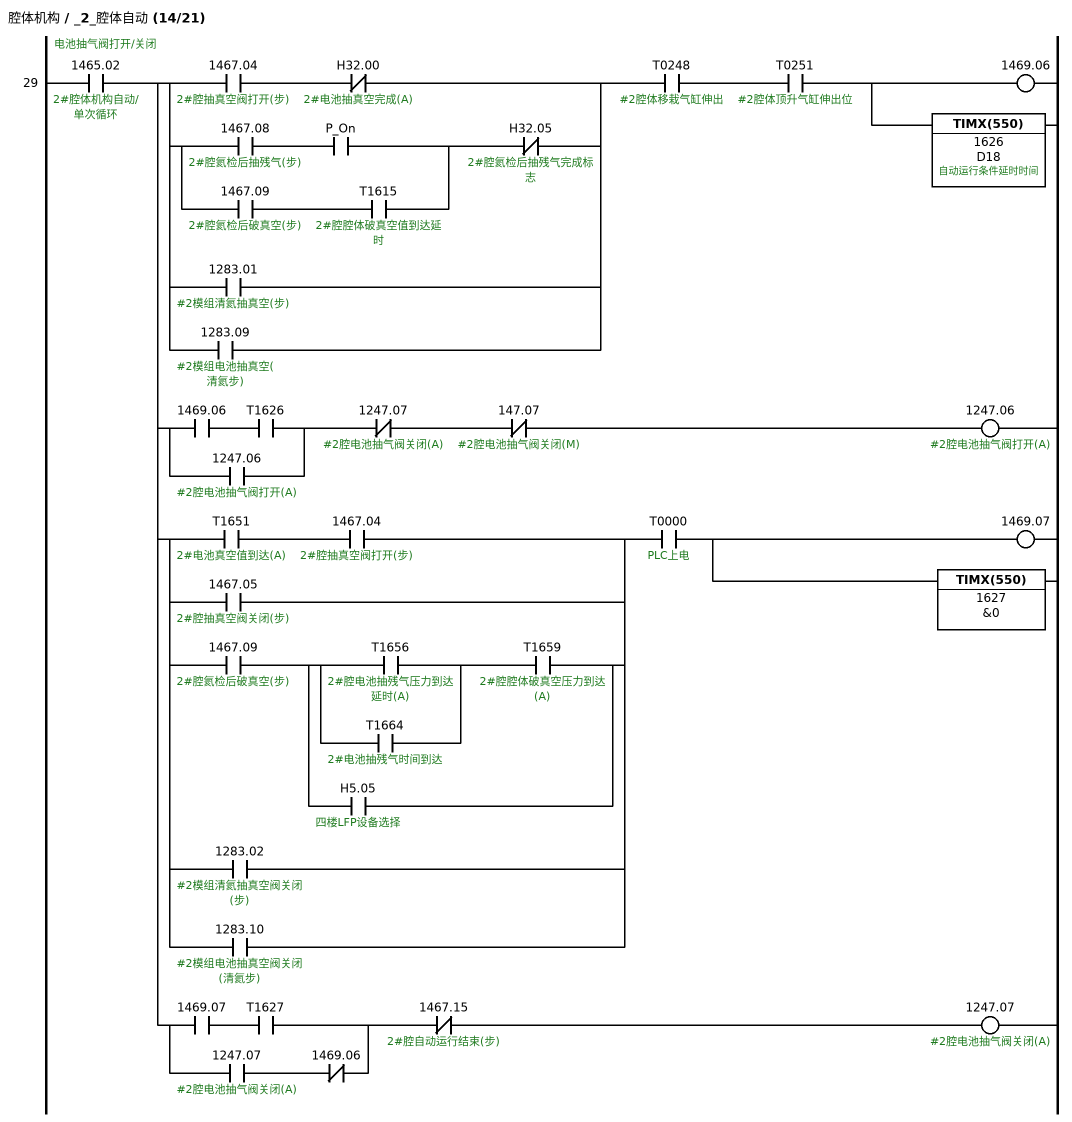
; [picture p312: 腔体机构 / _2_腔体自动, rungs 29-29]
; rung 29: 电池抽气阀打开/关闭
LD 1465.02  ; 2#腔体机构自动/单次循环
OUT TR0
LD 1467.04  ; 2#腔抽真空阀打开(步)
ANDNOT H32.00  ; 2#电池抽真空完成(A)
LD 1467.08  ; 2#腔氦检后抽残气(步)
AND P_On
LD 1467.09  ; 2#腔氦检后破真空(步)
AND T1615  ; 2#腔腔体破真空值到达延时
ORLD
ANDNOT H32.05  ; 2#腔氦检后抽残气完成标志
ORLD
OR 1283.01  ; #2模组清氦抽真空(步)
OR 1283.09  ; #2模组电池抽真空(清氦步)
ANDLD
AND T0248  ; #2腔体移栽气缸伸出
AND T0251  ; #2腔体顶升气缸伸出位
OUT 1469.06
TIMX(550) 1626 D18  ; 自动运行条件延时时间
LD TR0
LD 1469.06
AND T1626
OR 1247.06  ; #2腔电池抽气阀打开(A)
ANDLD
ANDNOT 1247.07  ; #2腔电池抽气阀关闭(A)
ANDNOT 147.07  ; #2腔电池抽气阀关闭(M)
OUT 1247.06  ; #2腔电池抽气阀打开(A)
LD TR0
LD T1651  ; 2#电池真空值到达(A)
AND 1467.04  ; 2#腔抽真空阀打开(步)
OR 1467.05  ; 2#腔抽真空阀关闭(步)
LD 1467.09  ; 2#腔氦检后破真空(步)
LD T1656  ; 2#腔电池抽残气压力到达延时(A)
OR T1664  ; 2#电池抽残气时间到达
AND T1659  ; 2#腔腔体破真空压力到达(A)
OR H5.05  ; 四楼LFP设备选择
ANDLD
ORLD
OR 1283.02  ; #2模组清氦抽真空阀关闭(步)
OR 1283.10  ; #2模组电池抽真空阀关闭(清氦步)
ANDLD
AND T0000  ; PLC上电
OUT 1469.07
TIMX(550) 1627 &0
LD TR0
LD 1469.07
AND T1627
LD 1247.07  ; #2腔电池抽气阀关闭(A)
ANDNOT 1469.06
ORLD
ANDLD
ANDNOT 1467.15  ; 2#腔自动运行结束(步)
OUT 1247.07  ; #2腔电池抽气阀关闭(A)

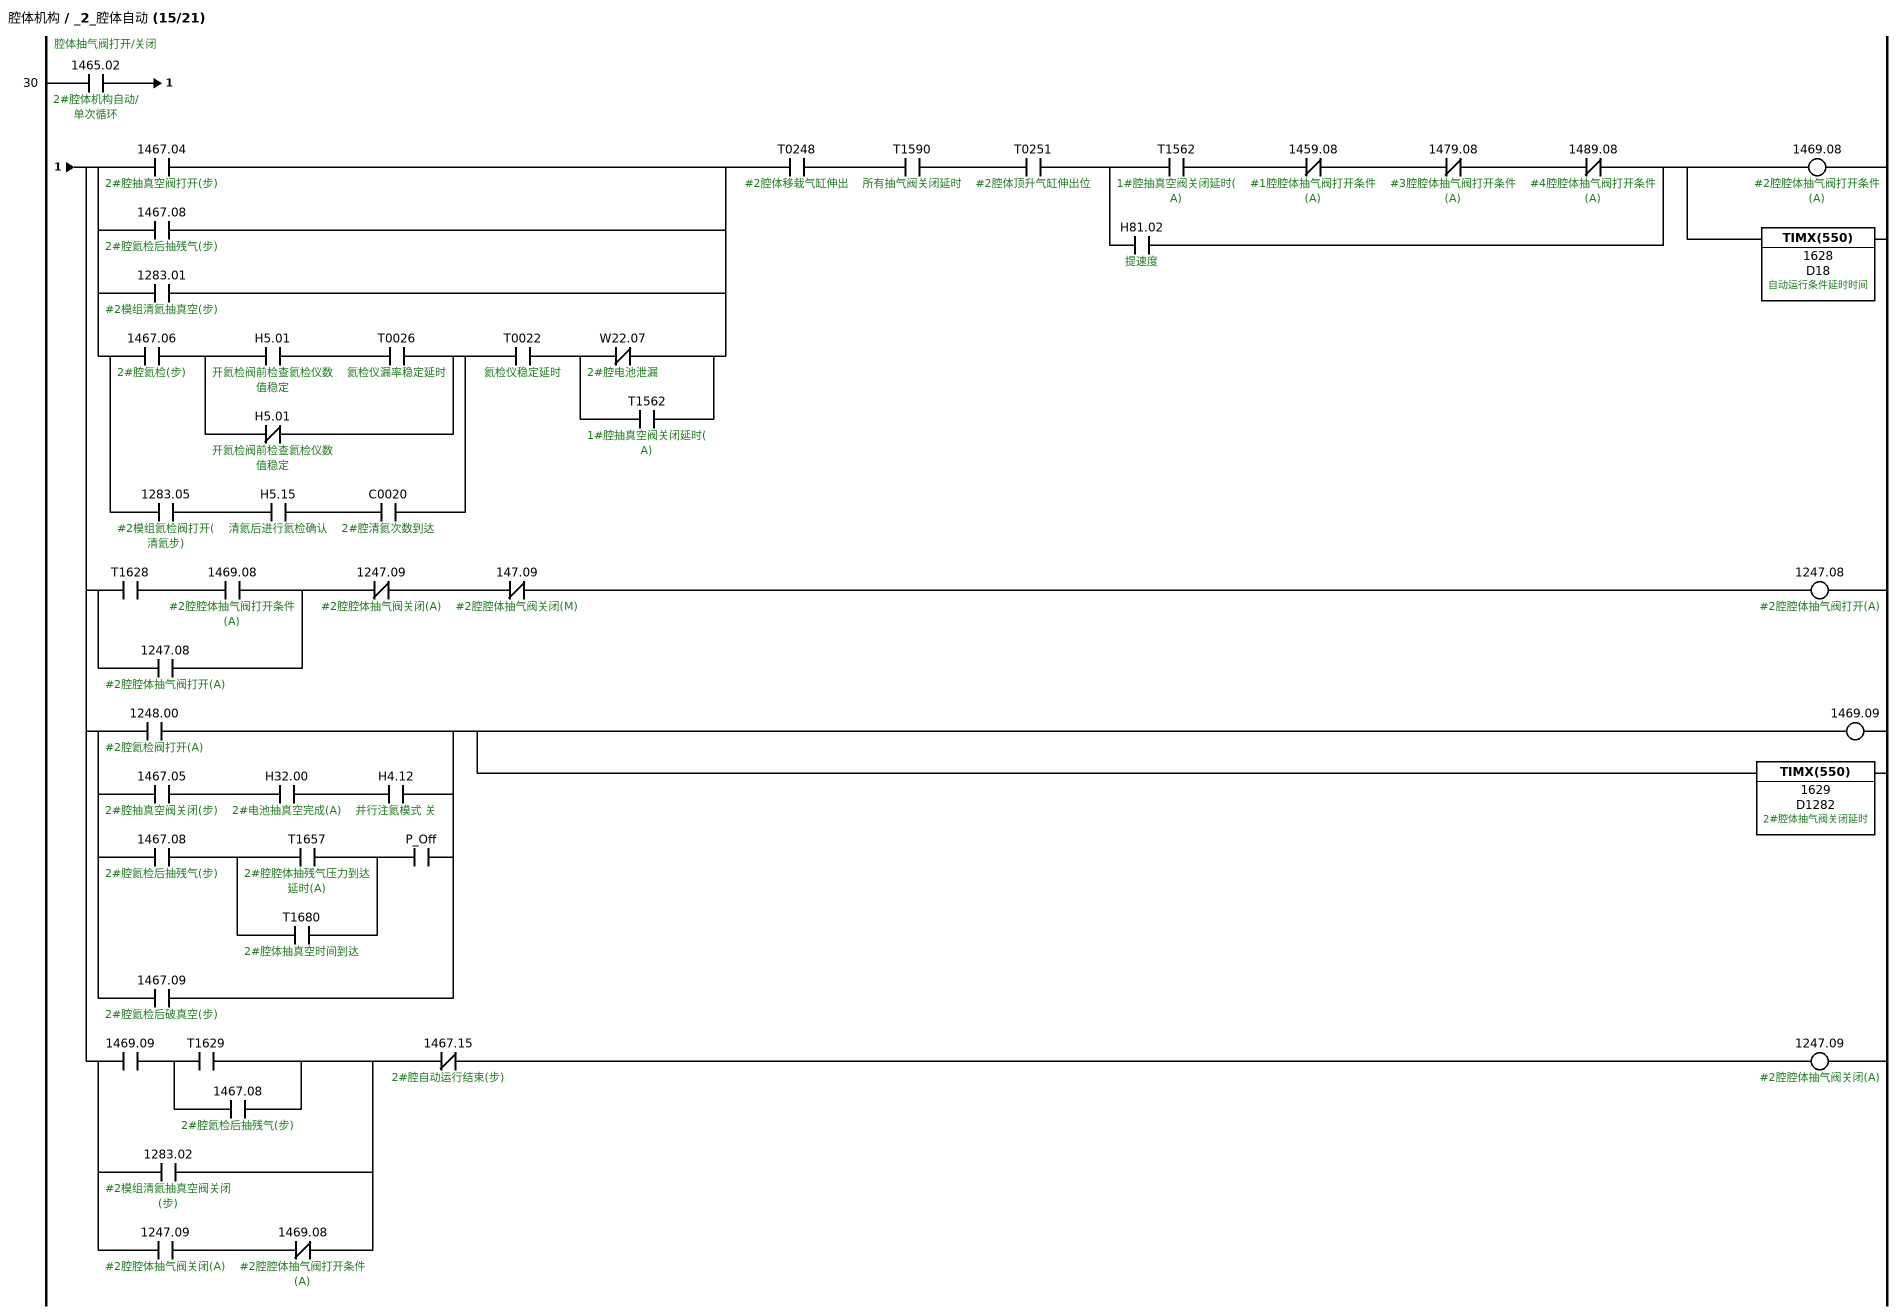
; rung 30: 腔体抽气阀打开/关闭
LD 1465.02  ; 2#腔体机构自动/单次循环
OUT TR0
LD 1467.04  ; 2#腔抽真空阀打开(步)
OR 1467.08  ; 2#腔氦检后抽残气(步)
OR 1283.01  ; #2模组清氦抽真空(步)
LD 1467.06  ; 2#腔氦检(步)
LD H5.01  ; 开氦检阀前检查氦检仪数值稳定
AND T0026  ; 氦检仪漏率稳定延时
ORNOT H5.01  ; 开氦检阀前检查氦检仪数值稳定
ANDLD
LD 1283.05  ; #2模组氦检阀打开(清氦步)
AND H5.15  ; 清氦后进行氦检确认
AND C0020  ; 2#腔清氦次数到达
ORLD
AND T0022  ; 氦检仪稳定延时
LDNOT W22.07  ; 2#腔电池泄漏
OR T1562  ; 1#腔抽真空阀关闭延时(A)
ANDLD
ORLD
ANDLD
AND T0248  ; #2腔体移栽气缸伸出
AND T1590  ; 所有抽气阀关闭延时
AND T0251  ; #2腔体顶升气缸伸出位
LD T1562  ; 1#腔抽真空阀关闭延时(A)
ANDNOT 1459.08  ; #1腔腔体抽气阀打开条件(A)
ANDNOT 1479.08  ; #3腔腔体抽气阀打开条件(A)
ANDNOT 1489.08  ; #4腔腔体抽气阀打开条件(A)
OR H81.02  ; 提速度
ANDLD
OUT 1469.08  ; #2腔腔体抽气阀打开条件(A)
TIMX(550) 1628 D18  ; 自动运行条件延时时间
LD TR0
LD T1628
AND 1469.08  ; #2腔腔体抽气阀打开条件(A)
OR 1247.08  ; #2腔腔体抽气阀打开(A)
ANDLD
ANDNOT 1247.09  ; #2腔腔体抽气阀关闭(A)
ANDNOT 147.09  ; #2腔腔体抽气阀关闭(M)
OUT 1247.08  ; #2腔腔体抽气阀打开(A)
LD TR0
LD 1248.00  ; #2腔氦检阀打开(A)
LD 1467.05  ; 2#腔抽真空阀关闭(步)
AND H32.00  ; 2#电池抽真空完成(A)
AND H4.12  ; 并行注氦模式 关
ORLD
LD 1467.08  ; 2#腔氦检后抽残气(步)
LD T1657  ; 2#腔腔体抽残气压力到达延时(A)
OR T1680  ; 2#腔体抽真空时间到达
ANDLD
AND P_Off
ORLD
OR 1467.09  ; 2#腔氦检后破真空(步)
ANDLD
OUT 1469.09
TIMX(550) 1629 D1282  ; 2#腔体抽气阀关闭延时
LD TR0
LD 1469.09
LD T1629
OR 1467.08  ; 2#腔氦检后抽残气(步)
ANDLD
OR 1283.02  ; #2模组清氦抽真空阀关闭(步)
LD 1247.09  ; #2腔腔体抽气阀关闭(A)
ANDNOT 1469.08  ; #2腔腔体抽气阀打开条件(A)
ORLD
ANDLD
ANDNOT 1467.15  ; 2#腔自动运行结束(步)
OUT 1247.09  ; #2腔腔体抽气阀关闭(A)

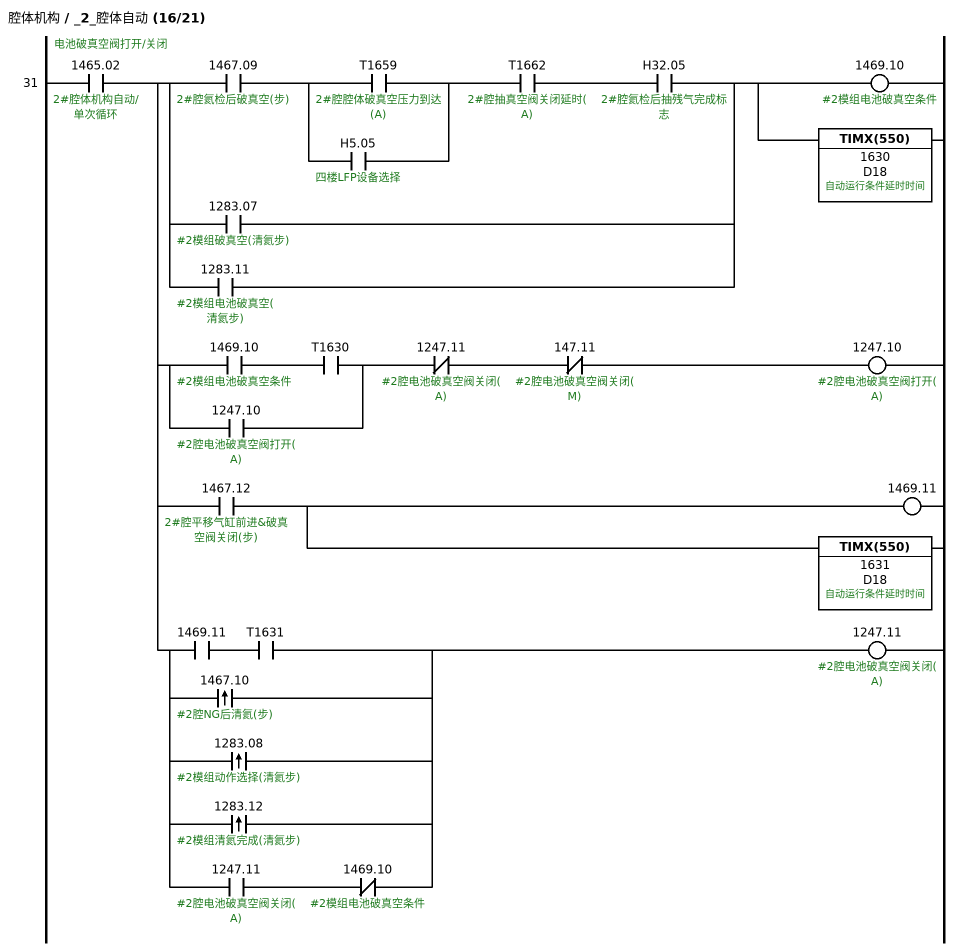
; rung 31: 电池破真空阀打开/关闭
LD 1465.02  ; 2#腔体机构自动/单次循环
OUT TR0
LD 1467.09  ; 2#腔氦检后破真空(步)
LD T1659  ; 2#腔腔体破真空压力到达(A)
OR H5.05  ; 四楼LFP设备选择
ANDLD
AND T1662  ; 2#腔抽真空阀关闭延时(A)
AND H32.05  ; 2#腔氦检后抽残气完成标志
OR 1283.07  ; #2模组破真空(清氦步)
OR 1283.11  ; #2模组电池破真空(清氦步)
ANDLD
OUT 1469.10  ; #2模组电池破真空条件
TIMX(550) 1630 D18  ; 自动运行条件延时时间
LD TR0
LD 1469.10  ; #2模组电池破真空条件
AND T1630
OR 1247.10  ; #2腔电池破真空阀打开(A)
ANDLD
ANDNOT 1247.11  ; #2腔电池破真空阀关闭(A)
ANDNOT 147.11  ; #2腔电池破真空阀关闭(M)
OUT 1247.10  ; #2腔电池破真空阀打开(A)
LD TR0
AND 1467.12  ; 2#腔平移气缸前进&破真空阀关闭(步)
OUT 1469.11
TIMX(550) 1631 D18  ; 自动运行条件延时时间
LD TR0
LD 1469.11
AND T1631
@OR 1467.10  ; #2腔NG后清氦(步)
@OR 1283.08  ; #2模组动作选择(清氦步)
@OR 1283.12  ; #2模组清氦完成(清氦步)
LD 1247.11  ; #2腔电池破真空阀关闭(A)
ANDNOT 1469.10  ; #2模组电池破真空条件
ORLD
ANDLD
OUT 1247.11  ; #2腔电池破真空阀关闭(A)

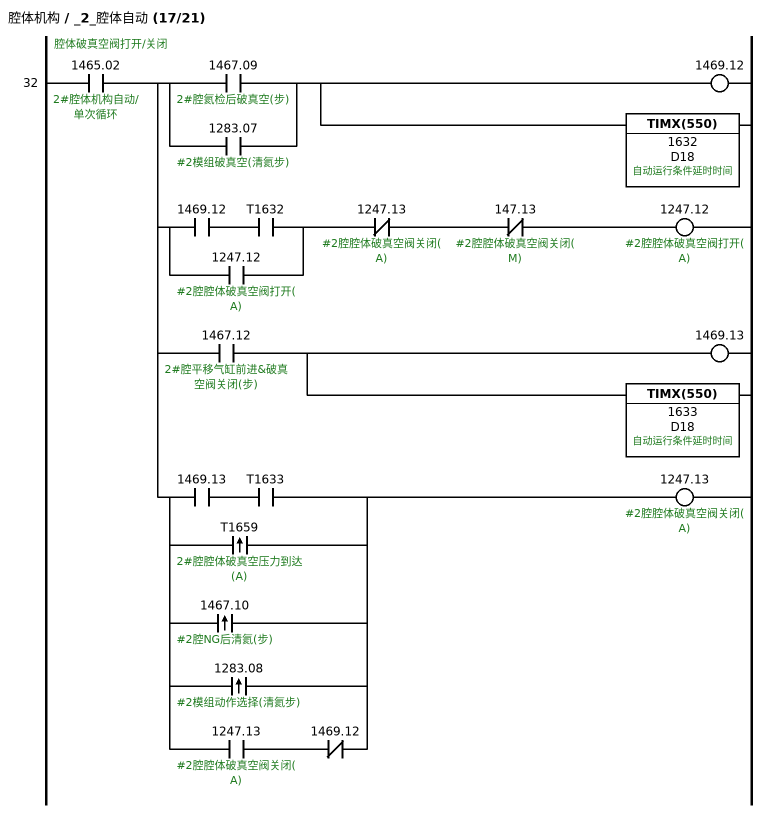
; rung 32: 腔体破真空阀打开/关闭
LD 1465.02  ; 2#腔体机构自动/单次循环
OUT TR0
LD 1467.09  ; 2#腔氦检后破真空(步)
OR 1283.07  ; #2模组破真空(清氦步)
ANDLD
OUT 1469.12
TIMX(550) 1632 D18  ; 自动运行条件延时时间
LD TR0
LD 1469.12
AND T1632
OR 1247.12  ; #2腔腔体破真空阀打开(A)
ANDLD
ANDNOT 1247.13  ; #2腔腔体破真空阀关闭(A)
ANDNOT 147.13  ; #2腔腔体破真空阀关闭(M)
OUT 1247.12  ; #2腔腔体破真空阀打开(A)
LD TR0
AND 1467.12  ; 2#腔平移气缸前进&破真空阀关闭(步)
OUT 1469.13
TIMX(550) 1633 D18  ; 自动运行条件延时时间
LD TR0
LD 1469.13
AND T1633
@OR T1659  ; 2#腔腔体破真空压力到达(A)
@OR 1467.10  ; #2腔NG后清氦(步)
@OR 1283.08  ; #2模组动作选择(清氦步)
LD 1247.13  ; #2腔腔体破真空阀关闭(A)
ANDNOT 1469.12
ORLD
ANDLD
OUT 1247.13  ; #2腔腔体破真空阀关闭(A)

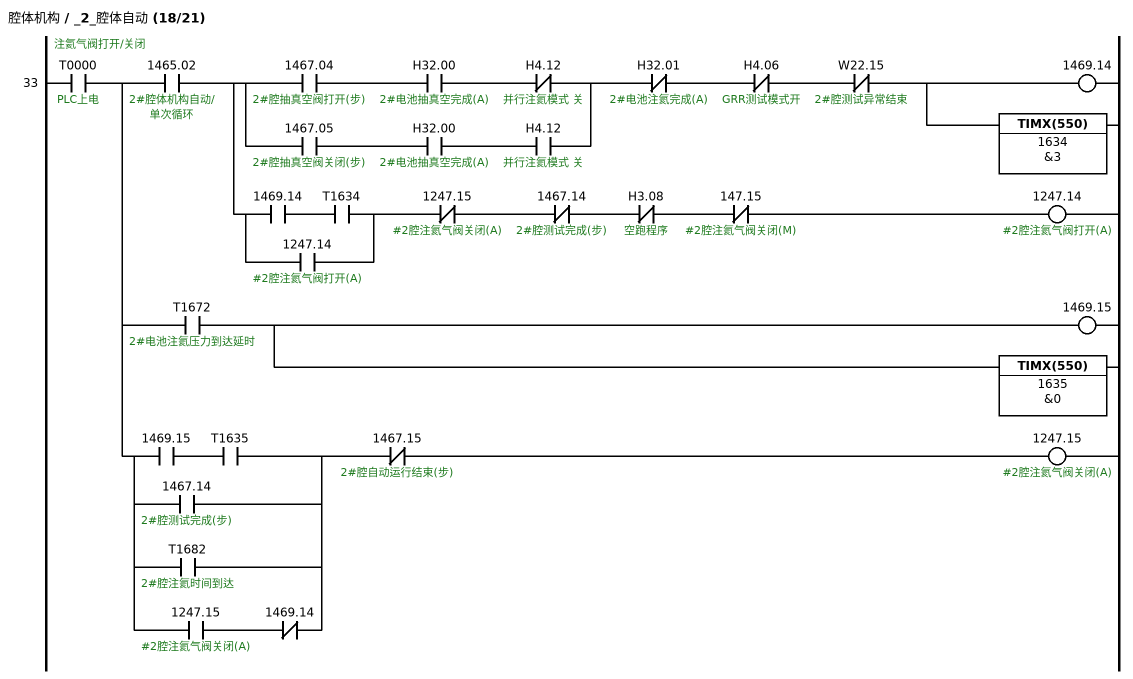
; rung 33: 注氦气阀打开/关闭
LD T0000  ; PLC上电
OUT TR0
AND 1465.02  ; 2#腔体机构自动/单次循环
OUT TR1
LD 1467.04  ; 2#腔抽真空阀打开(步)
AND H32.00  ; 2#电池抽真空完成(A)
ANDNOT H4.12  ; 并行注氦模式 关
LD 1467.05  ; 2#腔抽真空阀关闭(步)
AND H32.00  ; 2#电池抽真空完成(A)
AND H4.12  ; 并行注氦模式 关
ORLD
ANDLD
ANDNOT H32.01  ; 2#电池注氦完成(A)
ANDNOT H4.06  ; GRR测试模式开
ANDNOT W22.15  ; 2#腔测试异常结束
OUT 1469.14
TIMX(550) 1634 &3
LD TR1
LD 1469.14
AND T1634
OR 1247.14  ; #2腔注氦气阀打开(A)
ANDLD
ANDNOT 1247.15  ; #2腔注氦气阀关闭(A)
ANDNOT 1467.14  ; 2#腔测试完成(步)
ANDNOT H3.08  ; 空跑程序
ANDNOT 147.15  ; #2腔注氦气阀关闭(M)
OUT 1247.14  ; #2腔注氦气阀打开(A)
LD TR0
AND T1672  ; 2#电池注氦压力到达延时
OUT 1469.15
TIMX(550) 1635 &0
LD TR0
LD 1469.15
AND T1635
OR 1467.14  ; 2#腔测试完成(步)
OR T1682  ; 2#腔注氦时间到达
LD 1247.15  ; #2腔注氦气阀关闭(A)
ANDNOT 1469.14
ORLD
ANDLD
ANDNOT 1467.15  ; 2#腔自动运行结束(步)
OUT 1247.15  ; #2腔注氦气阀关闭(A)

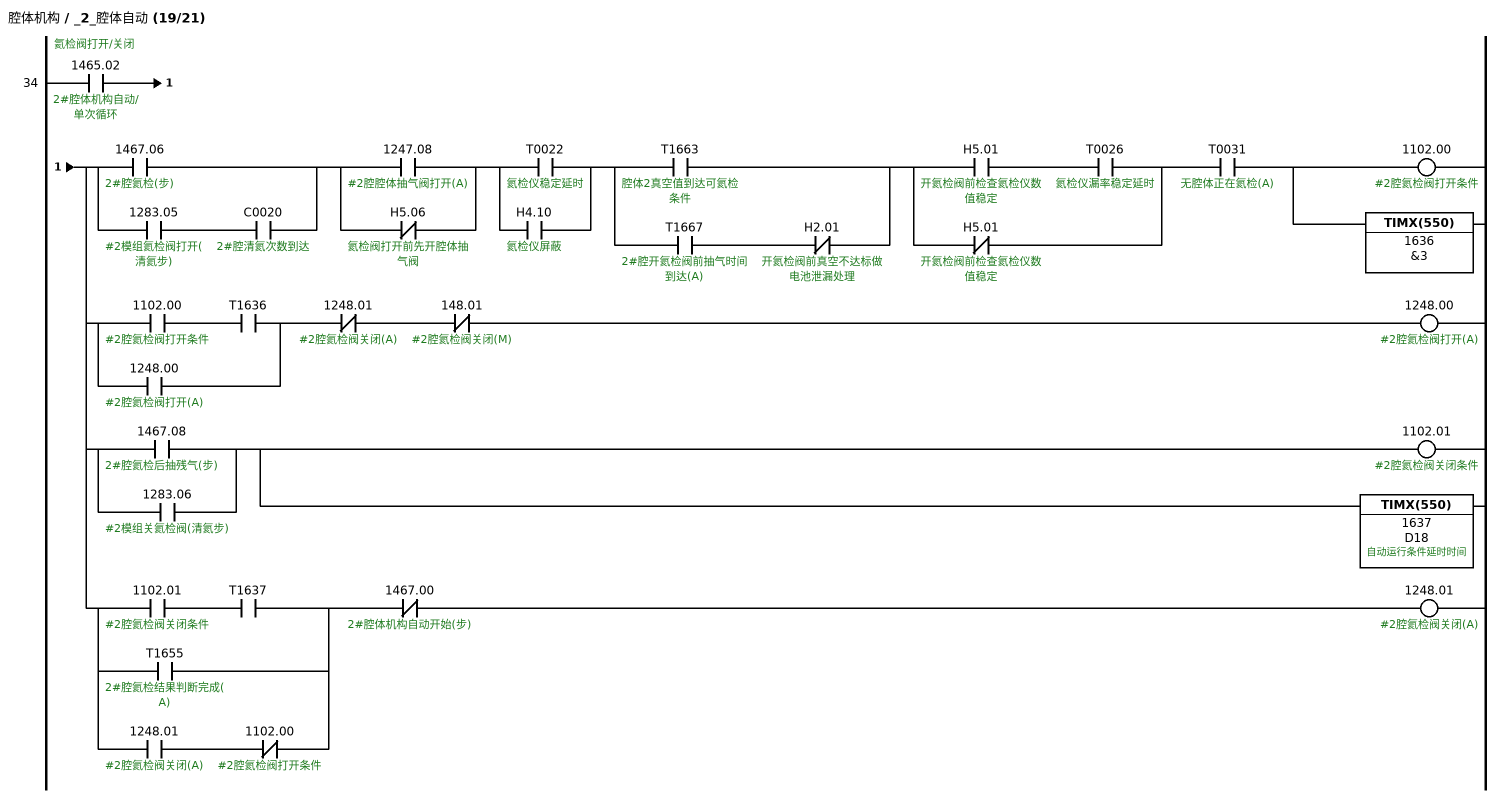
; rung 34: 氦检阀打开/关闭
LD 1465.02  ; 2#腔体机构自动/单次循环
OUT TR0
LD 1467.06  ; 2#腔氦检(步)
LD 1283.05  ; #2模组氦检阀打开(清氦步)
AND C0020  ; 2#腔清氦次数到达
ORLD
ANDLD
LD 1247.08  ; #2腔腔体抽气阀打开(A)
ORNOT H5.06  ; 氦检阀打开前先开腔体抽气阀
ANDLD
LD T0022  ; 氦检仪稳定延时
OR H4.10  ; 氦检仪屏蔽
ANDLD
LD T1663  ; 腔体2真空值到达可氦检条件
LD T1667  ; 2#腔开氦检阀前抽气时间到达(A)
ANDNOT H2.01  ; 开氦检阀前真空不达标做电池泄漏处理
ORLD
ANDLD
LD H5.01  ; 开氦检阀前检查氦检仪数值稳定
AND T0026  ; 氦检仪漏率稳定延时
ORNOT H5.01  ; 开氦检阀前检查氦检仪数值稳定
ANDLD
AND T0031  ; 无腔体正在氦检(A)
OUT 1102.00  ; #2腔氦检阀打开条件
TIMX(550) 1636 &3
LD TR0
LD 1102.00  ; #2腔氦检阀打开条件
AND T1636
OR 1248.00  ; #2腔氦检阀打开(A)
ANDLD
ANDNOT 1248.01  ; #2腔氦检阀关闭(A)
ANDNOT 148.01  ; #2腔氦检阀关闭(M)
OUT 1248.00  ; #2腔氦检阀打开(A)
LD TR0
LD 1467.08  ; 2#腔氦检后抽残气(步)
OR 1283.06  ; #2模组关氦检阀(清氦步)
ANDLD
OUT 1102.01  ; #2腔氦检阀关闭条件
TIMX(550) 1637 D18  ; 自动运行条件延时时间
LD TR0
LD 1102.01  ; #2腔氦检阀关闭条件
AND T1637
OR T1655  ; 2#腔氦检结果判断完成(A)
LD 1248.01  ; #2腔氦检阀关闭(A)
ANDNOT 1102.00  ; #2腔氦检阀打开条件
ORLD
ANDLD
ANDNOT 1467.00  ; 2#腔体机构自动开始(步)
OUT 1248.01  ; #2腔氦检阀关闭(A)

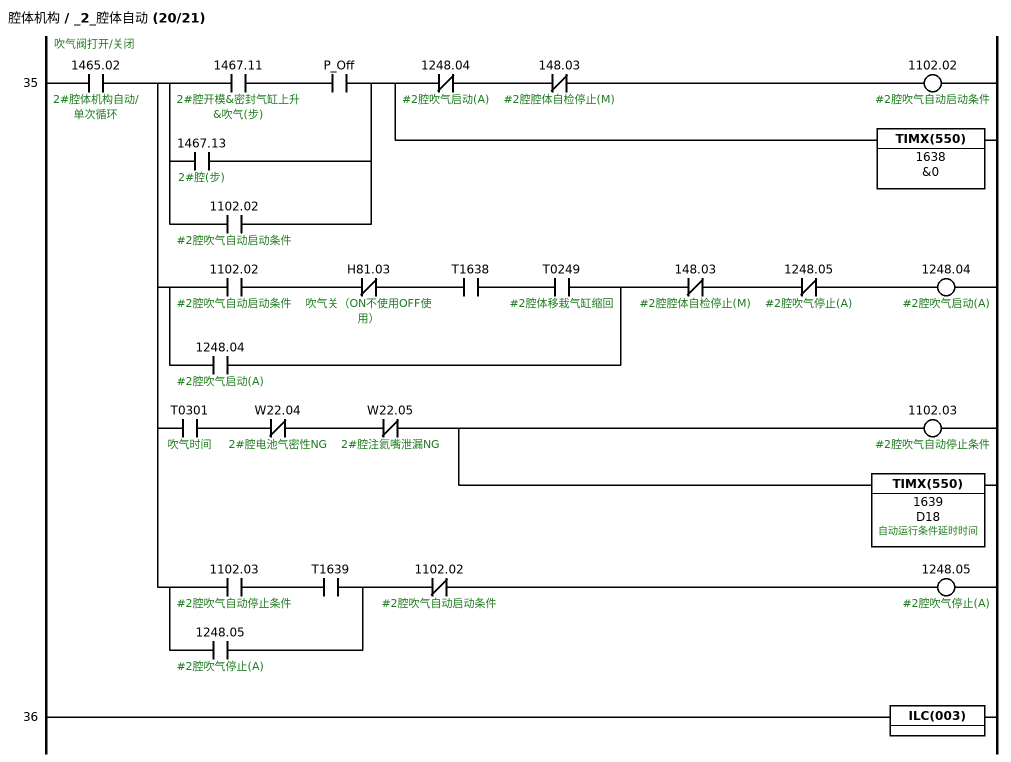
; rung 35: 吹气阀打开/关闭
LD 1465.02  ; 2#腔体机构自动/单次循环
OUT TR0
LD 1467.11  ; 2#腔开模&密封气缸上升&吹气(步)
AND P_Off
OR 1467.13  ; 2#腔(步)
OR 1102.02  ; #2腔吹气自动启动条件
ANDLD
OUT TR1
ANDNOT 1248.04  ; #2腔吹气启动(A)
ANDNOT 148.03  ; #2腔腔体自检停止(M)
OUT 1102.02  ; #2腔吹气自动启动条件
LD TR1
TIMX(550) 1638 &0
LD TR0
LD 1102.02  ; #2腔吹气自动启动条件
ANDNOT H81.03  ; 吹气关（ON不使用OFF使用）
AND T1638
AND T0249  ; #2腔体移栽气缸缩回
OR 1248.04  ; #2腔吹气启动(A)
ANDLD
ANDNOT 148.03  ; #2腔腔体自检停止(M)
ANDNOT 1248.05  ; #2腔吹气停止(A)
OUT 1248.04  ; #2腔吹气启动(A)
LD TR0
AND T0301  ; 吹气时间
ANDNOT W22.04  ; 2#腔电池气密性NG
ANDNOT W22.05  ; 2#腔注氦嘴泄漏NG
OUT 1102.03  ; #2腔吹气自动停止条件
TIMX(550) 1639 D18  ; 自动运行条件延时时间
LD TR0
LD 1102.03  ; #2腔吹气自动停止条件
AND T1639
OR 1248.05  ; #2腔吹气停止(A)
ANDLD
ANDNOT 1102.02  ; #2腔吹气自动启动条件
OUT 1248.05  ; #2腔吹气停止(A)
; rung 36
ILC(003)

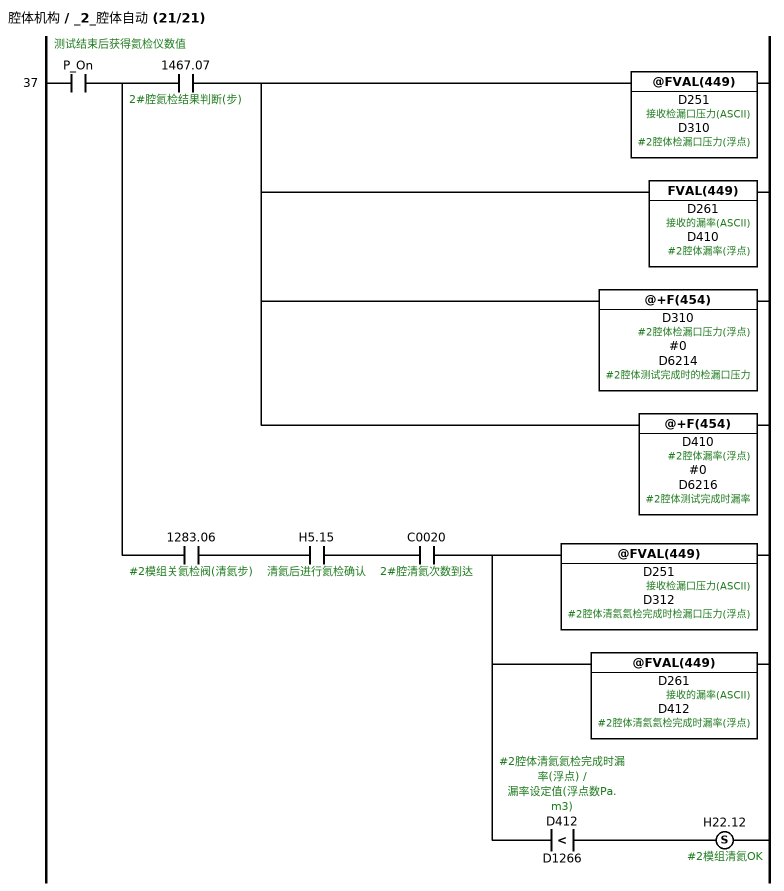
; rung 37: 测试结束后获得氦检仪数值
LD P_On
OUT TR0
AND 1467.07  ; 2#腔氦检结果判断(步)
@FVAL(449) D251 D310  ; 接收检漏口压力(ASCII), #2腔体检漏口压力(浮点)
FVAL(449) D261 D410  ; 接收的漏率(ASCII), #2腔体漏率(浮点)
@+F(454) D310 #0 D6214  ; #2腔体检漏口压力(浮点), #2腔体测试完成时的检漏口压力
@+F(454) D410 #0 D6216  ; #2腔体漏率(浮点), #2腔体测试完成时漏率
LD TR0
AND 1283.06  ; #2模组关氦检阀(清氦步)
AND H5.15  ; 清氦后进行氦检确认
AND C0020  ; 2#腔清氦次数到达
@FVAL(449) D251 D312  ; 接收检漏口压力(ASCII), #2腔体清氦氦检完成时检漏口压力(浮点)
@FVAL(449) D261 D412  ; 接收的漏率(ASCII), #2腔体清氦氦检完成时漏率(浮点)
AND<F(331) D412 D1266  ; #2腔体清氦氦检完成时漏率(浮点), 漏率设定值(浮点数Pa.m3)
SET H22.12  ; #2模组清氦OK

### Section _3_腔体自动

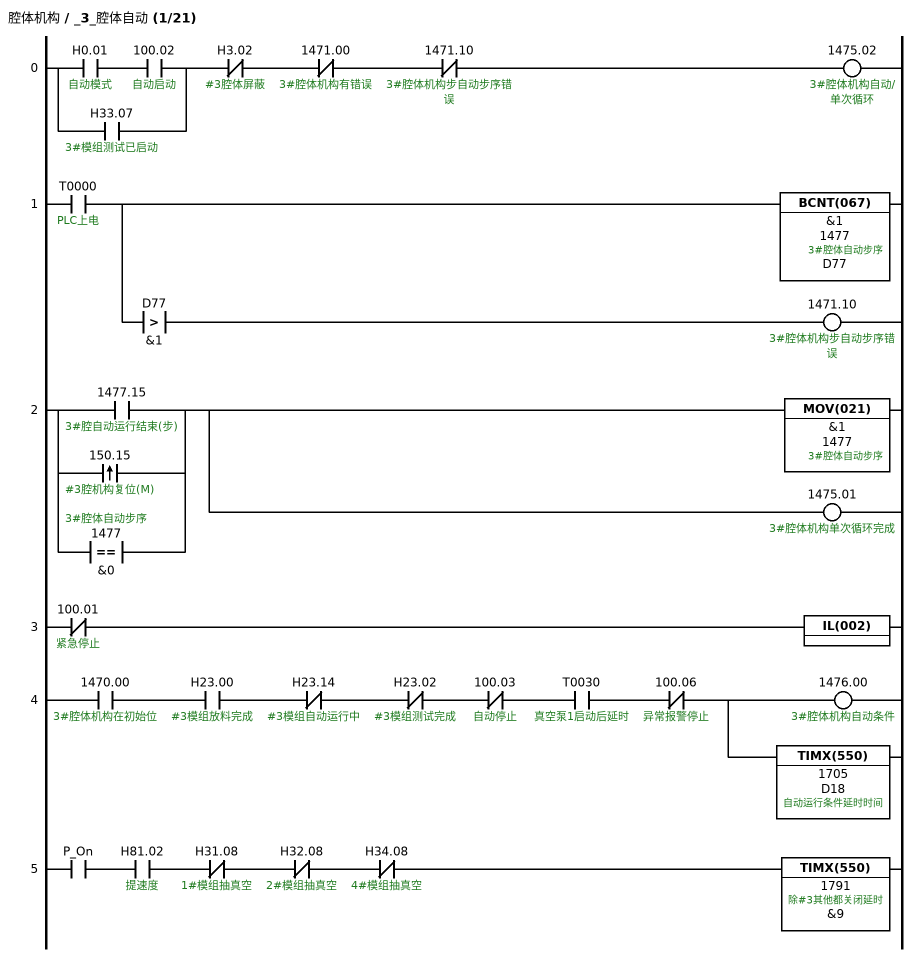
; rung 0
LD H0.01  ; 自动模式
AND 100.02  ; 自动启动
OR H33.07  ; 3#模组测试已启动
ANDNOT H3.02  ; #3腔体屏蔽
ANDNOT 1471.00  ; 3#腔体机构有错误
ANDNOT 1471.10  ; 3#腔体机构步自动步序错误
OUT 1475.02  ; 3#腔体机构自动/单次循环
; rung 1
LD T0000  ; PLC上电
BCNT(067) &1 1477 D77  ; 3#腔体自动步序
AND>(320) D77 &1
OUT 1471.10  ; 3#腔体机构步自动步序错误
; rung 2
LD 1477.15  ; 3#腔自动运行结束(步)
@OR 150.15  ; #3腔机构复位(M)
OR=(300) 1477 &0  ; 3#腔体自动步序
MOV(021) &1 1477  ; 3#腔体自动步序
OUT 1475.01  ; 3#腔体机构单次循环完成
; rung 3
LDNOT 100.01  ; 紧急停止
IL(002)
; rung 4
LD 1470.00  ; 3#腔体机构在初始位
AND H23.00  ; #3模组放料完成
ANDNOT H23.14  ; #3模组自动运行中
ANDNOT H23.02  ; #3模组测试完成
ANDNOT 100.03  ; 自动停止
AND T0030  ; 真空泵1启动后延时
ANDNOT 100.06  ; 异常报警停止
OUT 1476.00  ; 3#腔体机构自动条件
TIMX(550) 1705 D18  ; 自动运行条件延时时间
; rung 5
LD P_On
AND H81.02  ; 提速度
ANDNOT H31.08  ; 1#模组抽真空
ANDNOT H32.08  ; 2#模组抽真空
ANDNOT H34.08  ; 4#模组抽真空
TIMX(550) 1791 &9  ; 除#3其他都关闭延时

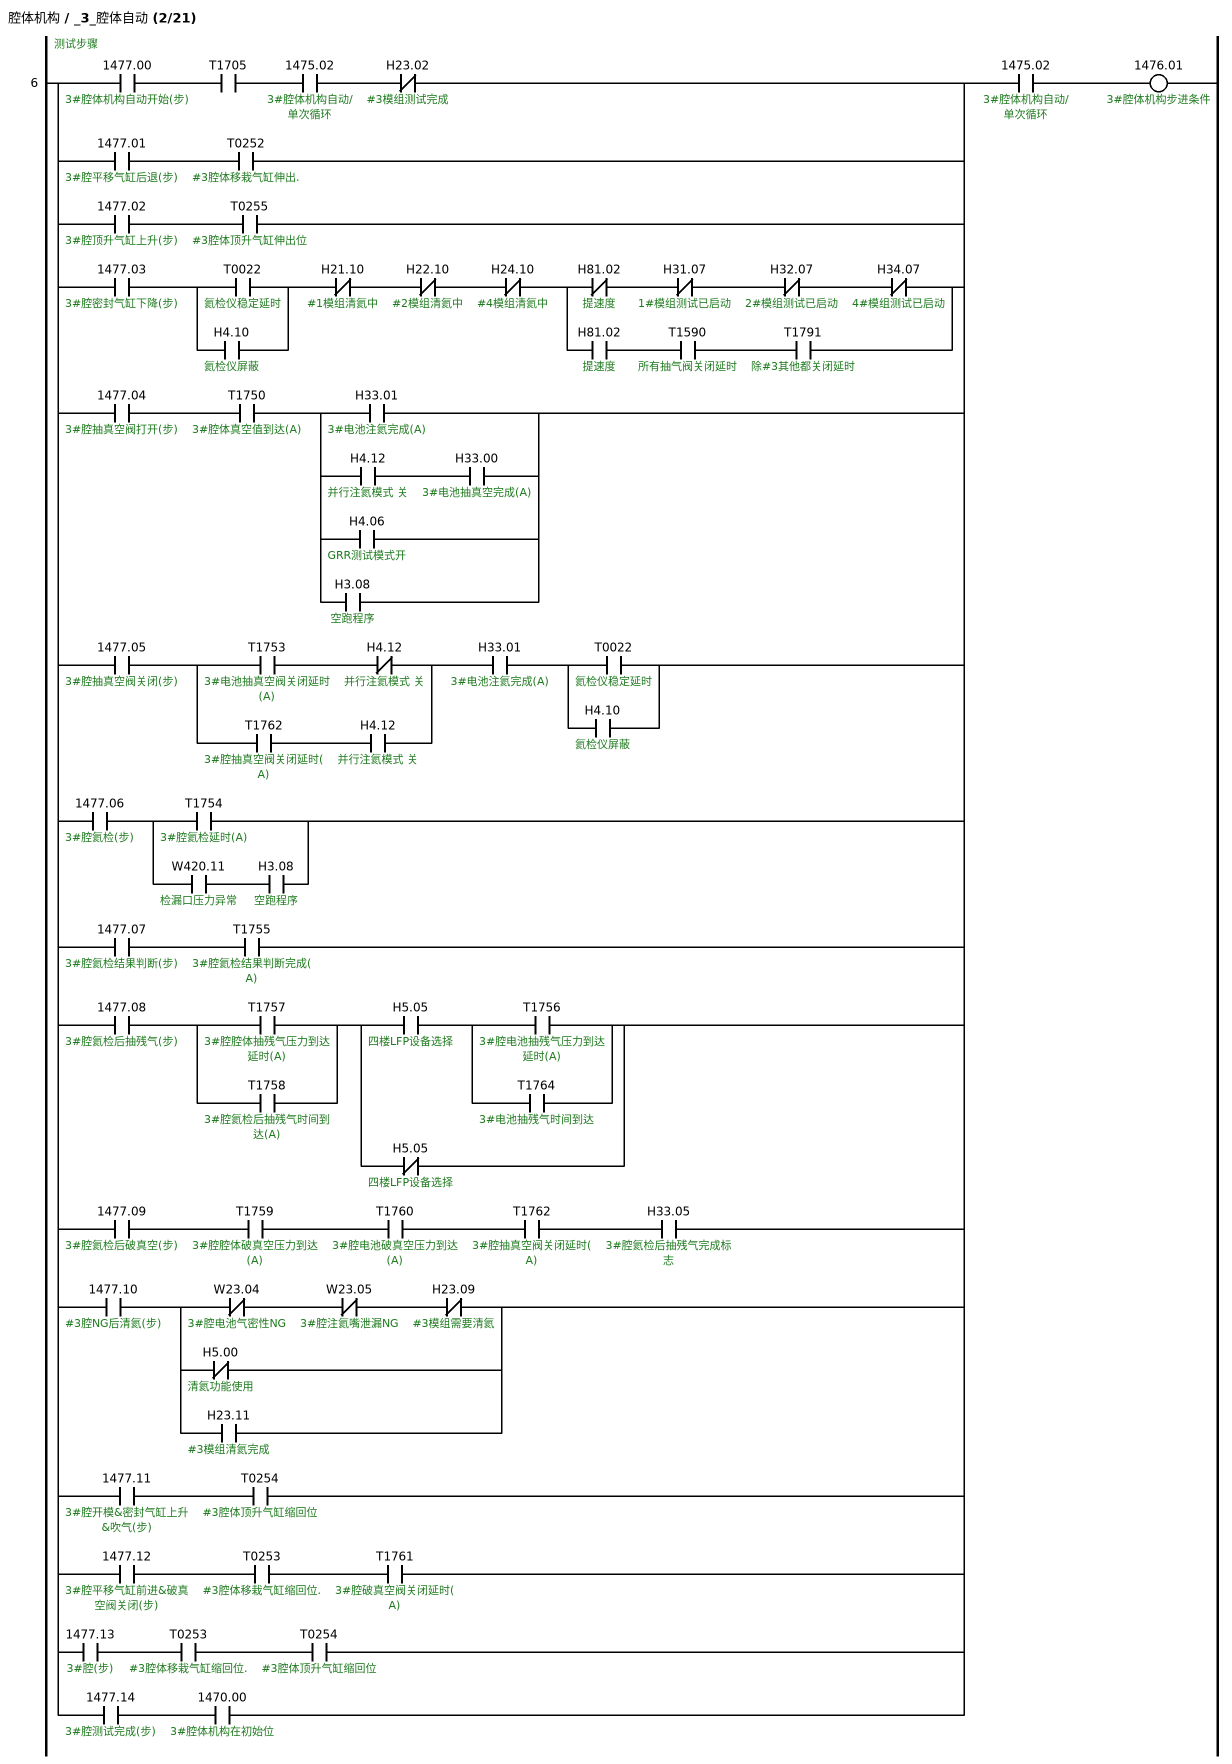
; rung 6: 测试步骤
LD 1477.00  ; 3#腔体机构自动开始(步)
AND T1705
AND 1475.02  ; 3#腔体机构自动/单次循环
ANDNOT H23.02  ; #3模组测试完成
LD 1477.01  ; 3#腔平移气缸后退(步)
AND T0252  ; #3腔体移栽气缸伸出.
ORLD
LD 1477.02  ; 3#腔顶升气缸上升(步)
AND T0255  ; #3腔体顶升气缸伸出位
ORLD
LD 1477.03  ; 3#腔密封气缸下降(步)
LD T0022  ; 氦检仪稳定延时
OR H4.10  ; 氦检仪屏蔽
ANDLD
ANDNOT H21.10  ; #1模组清氦中
ANDNOT H22.10  ; #2模组清氦中
ANDNOT H24.10  ; #4模组清氦中
LDNOT H81.02  ; 提速度
ANDNOT H31.07  ; 1#模组测试已启动
ANDNOT H32.07  ; 2#模组测试已启动
ANDNOT H34.07  ; 4#模组测试已启动
LD H81.02  ; 提速度
AND T1590  ; 所有抽气阀关闭延时
AND T1791  ; 除#3其他都关闭延时
ORLD
ANDLD
ORLD
LD 1477.04  ; 3#腔抽真空阀打开(步)
AND T1750  ; 3#腔体真空值到达(A)
LD H33.01  ; 3#电池注氦完成(A)
LD H4.12  ; 并行注氦模式 关
AND H33.00  ; 3#电池抽真空完成(A)
ORLD
OR H4.06  ; GRR测试模式开
OR H3.08  ; 空跑程序
ANDLD
ORLD
LD 1477.05  ; 3#腔抽真空阀关闭(步)
LD T1753  ; 3#电池抽真空阀关闭延时(A)
ANDNOT H4.12  ; 并行注氦模式 关
LD T1762  ; 3#腔抽真空阀关闭延时(A)
AND H4.12  ; 并行注氦模式 关
ORLD
ANDLD
AND H33.01  ; 3#电池注氦完成(A)
LD T0022  ; 氦检仪稳定延时
OR H4.10  ; 氦检仪屏蔽
ANDLD
ORLD
LD 1477.06  ; 3#腔氦检(步)
LD T1754  ; 3#腔氦检延时(A)
LD W420.11  ; 检漏口压力异常
AND H3.08  ; 空跑程序
ORLD
ANDLD
ORLD
LD 1477.07  ; 3#腔氦检结果判断(步)
AND T1755  ; 3#腔氦检结果判断完成(A)
ORLD
LD 1477.08  ; 3#腔氦检后抽残气(步)
LD T1757  ; 3#腔腔体抽残气压力到达延时(A)
OR T1758  ; 3#腔氦检后抽残气时间到达(A)
ANDLD
LD H5.05  ; 四楼LFP设备选择
LD T1756  ; 3#腔电池抽残气压力到达延时(A)
OR T1764  ; 3#电池抽残气时间到达
ANDLD
ORNOT H5.05  ; 四楼LFP设备选择
ANDLD
ORLD
LD 1477.09  ; 3#腔氦检后破真空(步)
AND T1759  ; 3#腔腔体破真空压力到达(A)
AND T1760  ; 3#腔电池破真空压力到达(A)
AND T1762  ; 3#腔抽真空阀关闭延时(A)
AND H33.05  ; 3#腔氦检后抽残气完成标志
ORLD
LD 1477.10  ; #3腔NG后清氦(步)
LDNOT W23.04  ; 3#腔电池气密性NG
ANDNOT W23.05  ; 3#腔注氦嘴泄漏NG
ANDNOT H23.09  ; #3模组需要清氦
ORNOT H5.00  ; 清氦功能使用
OR H23.11  ; #3模组清氦完成
ANDLD
ORLD
LD 1477.11  ; 3#腔开模&密封气缸上升&吹气(步)
AND T0254  ; #3腔体顶升气缸缩回位
ORLD
LD 1477.12  ; 3#腔平移气缸前进&破真空阀关闭(步)
AND T0253  ; #3腔体移栽气缸缩回位.
AND T1761  ; 3#腔破真空阀关闭延时(A)
ORLD
LD 1477.13  ; 3#腔(步)
AND T0253  ; #3腔体移栽气缸缩回位.
AND T0254  ; #3腔体顶升气缸缩回位
ORLD
LD 1477.14  ; 3#腔测试完成(步)
AND 1470.00  ; 3#腔体机构在初始位
ORLD
AND 1475.02  ; 3#腔体机构自动/单次循环
OUT 1476.01  ; 3#腔体机构步进条件

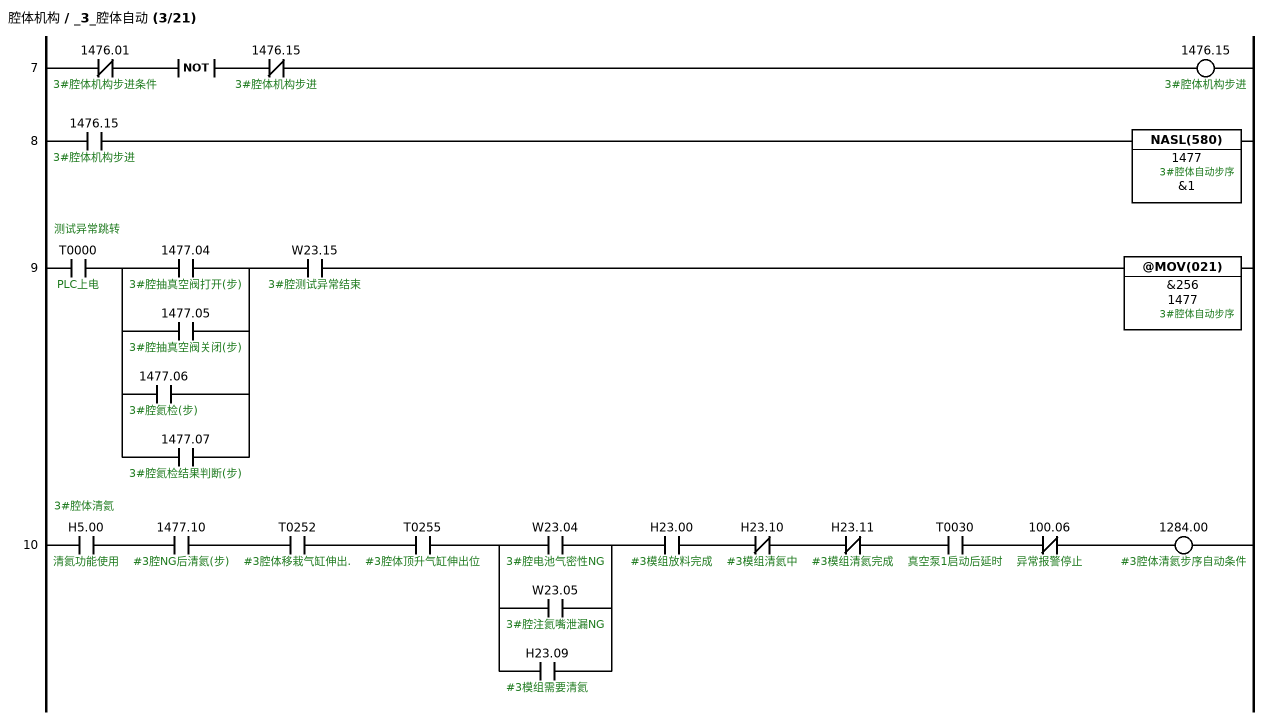
; rung 7
LDNOT 1476.01  ; 3#腔体机构步进条件
NOT(520)
ANDNOT 1476.15  ; 3#腔体机构步进
OUT 1476.15  ; 3#腔体机构步进
; rung 8
LD 1476.15  ; 3#腔体机构步进
NASL(580) 1477 &1  ; 3#腔体自动步序
; rung 9: 测试异常跳转
LD T0000  ; PLC上电
LD 1477.04  ; 3#腔抽真空阀打开(步)
OR 1477.05  ; 3#腔抽真空阀关闭(步)
OR 1477.06  ; 3#腔氦检(步)
OR 1477.07  ; 3#腔氦检结果判断(步)
ANDLD
AND W23.15  ; 3#腔测试异常结束
@MOV(021) &256 1477  ; 3#腔体自动步序
; rung 10: 3#腔体清氦
LD H5.00  ; 清氦功能使用
AND 1477.10  ; #3腔NG后清氦(步)
AND T0252  ; #3腔体移栽气缸伸出.
AND T0255  ; #3腔体顶升气缸伸出位
LD W23.04  ; 3#腔电池气密性NG
OR W23.05  ; 3#腔注氦嘴泄漏NG
OR H23.09  ; #3模组需要清氦
ANDLD
AND H23.00  ; #3模组放料完成
ANDNOT H23.10  ; #3模组清氦中
ANDNOT H23.11  ; #3模组清氦完成
AND T0030  ; 真空泵1启动后延时
ANDNOT 100.06  ; 异常报警停止
OUT 1284.00  ; #3腔体清氦步序自动条件

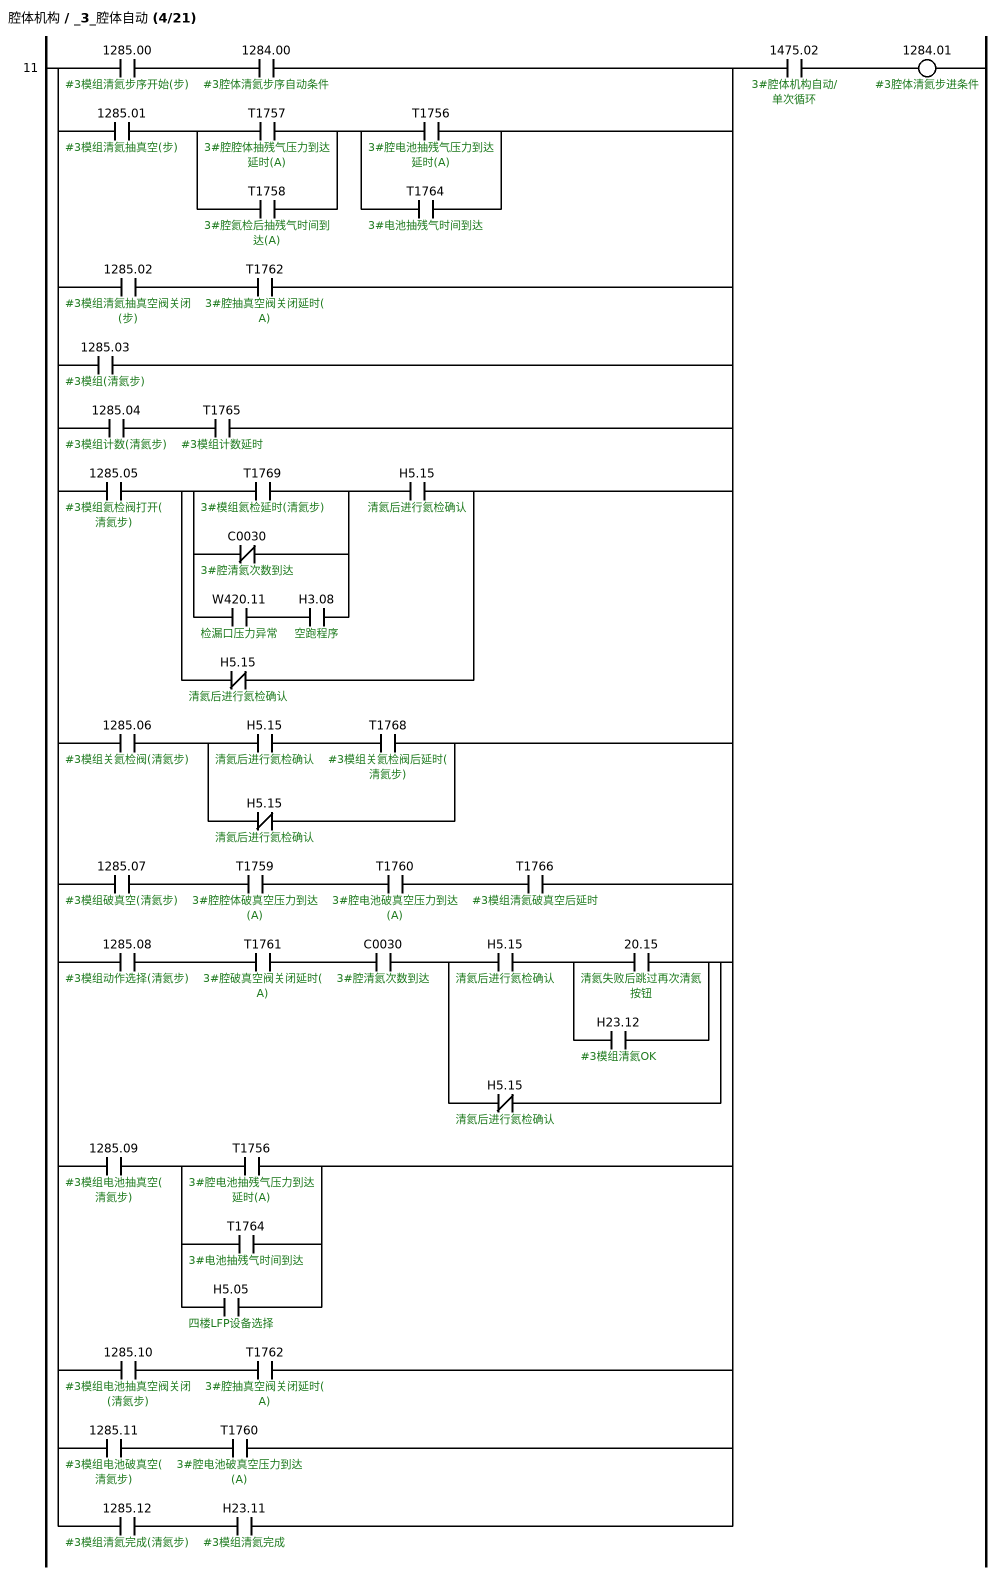
; rung 11
LD 1285.00  ; #3模组清氦步序开始(步)
AND 1284.00  ; #3腔体清氦步序自动条件
LD 1285.01  ; #3模组清氦抽真空(步)
LD T1757  ; 3#腔腔体抽残气压力到达延时(A)
OR T1758  ; 3#腔氦检后抽残气时间到达(A)
ANDLD
LD T1756  ; 3#腔电池抽残气压力到达延时(A)
OR T1764  ; 3#电池抽残气时间到达
ANDLD
ORLD
LD 1285.02  ; #3模组清氦抽真空阀关闭(步)
AND T1762  ; 3#腔抽真空阀关闭延时(A)
ORLD
OR 1285.03  ; #3模组(清氦步)
LD 1285.04  ; #3模组计数(清氦步)
AND T1765  ; #3模组计数延时
ORLD
LD 1285.05  ; #3模组氦检阀打开(清氦步)
LD T1769  ; 3#模组氦检延时(清氦步)
ORNOT C0030  ; 3#腔清氦次数到达
LD W420.11  ; 检漏口压力异常
AND H3.08  ; 空跑程序
ORLD
AND H5.15  ; 清氦后进行氦检确认
ORNOT H5.15  ; 清氦后进行氦检确认
ANDLD
ORLD
LD 1285.06  ; #3模组关氦检阀(清氦步)
LD H5.15  ; 清氦后进行氦检确认
AND T1768  ; #3模组关氦检阀后延时(清氦步)
ORNOT H5.15  ; 清氦后进行氦检确认
ANDLD
ORLD
LD 1285.07  ; #3模组破真空(清氦步)
AND T1759  ; 3#腔腔体破真空压力到达(A)
AND T1760  ; 3#腔电池破真空压力到达(A)
AND T1766  ; #3模组清氦破真空后延时
ORLD
LD 1285.08  ; #3模组动作选择(清氦步)
AND T1761  ; 3#腔破真空阀关闭延时(A)
AND C0030  ; 3#腔清氦次数到达
LD H5.15  ; 清氦后进行氦检确认
LD 20.15  ; 清氦失败后跳过再次清氦按钮
OR H23.12  ; #3模组清氦OK
ANDLD
ORNOT H5.15  ; 清氦后进行氦检确认
ANDLD
ORLD
LD 1285.09  ; #3模组电池抽真空(清氦步)
LD T1756  ; 3#腔电池抽残气压力到达延时(A)
OR T1764  ; 3#电池抽残气时间到达
OR H5.05  ; 四楼LFP设备选择
ANDLD
ORLD
LD 1285.10  ; #3模组电池抽真空阀关闭(清氦步)
AND T1762  ; 3#腔抽真空阀关闭延时(A)
ORLD
LD 1285.11  ; #3模组电池破真空(清氦步)
AND T1760  ; 3#腔电池破真空压力到达(A)
ORLD
LD 1285.12  ; #3模组清氦完成(清氦步)
AND H23.11  ; #3模组清氦完成
ORLD
AND 1475.02  ; 3#腔体机构自动/单次循环
OUT 1284.01  ; #3腔体清氦步进条件

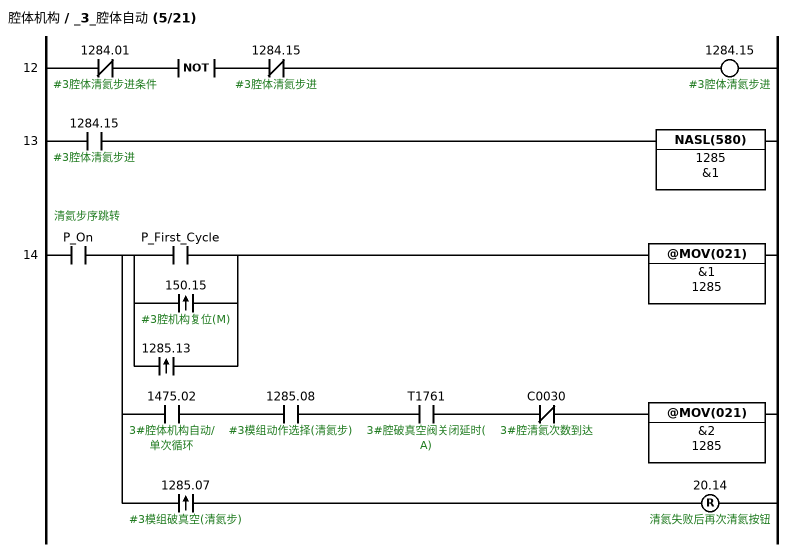
; rung 12
LDNOT 1284.01  ; #3腔体清氦步进条件
NOT(520)
ANDNOT 1284.15  ; #3腔体清氦步进
OUT 1284.15  ; #3腔体清氦步进
; rung 13
LD 1284.15  ; #3腔体清氦步进
NASL(580) 1285 &1
; rung 14: 清氦步序跳转
LD P_On
OUT TR0
LD P_First_Cycle
@OR 150.15  ; #3腔机构复位(M)
@OR 1285.13
ANDLD
@MOV(021) &1 1285
LD TR0
AND 1475.02  ; 3#腔体机构自动/单次循环
AND 1285.08  ; #3模组动作选择(清氦步)
AND T1761  ; 3#腔破真空阀关闭延时(A)
ANDNOT C0030  ; 3#腔清氦次数到达
@MOV(021) &2 1285
LD TR0
@AND 1285.07  ; #3模组破真空(清氦步)
RSET 20.14  ; 清氦失败后再次清氦按钮

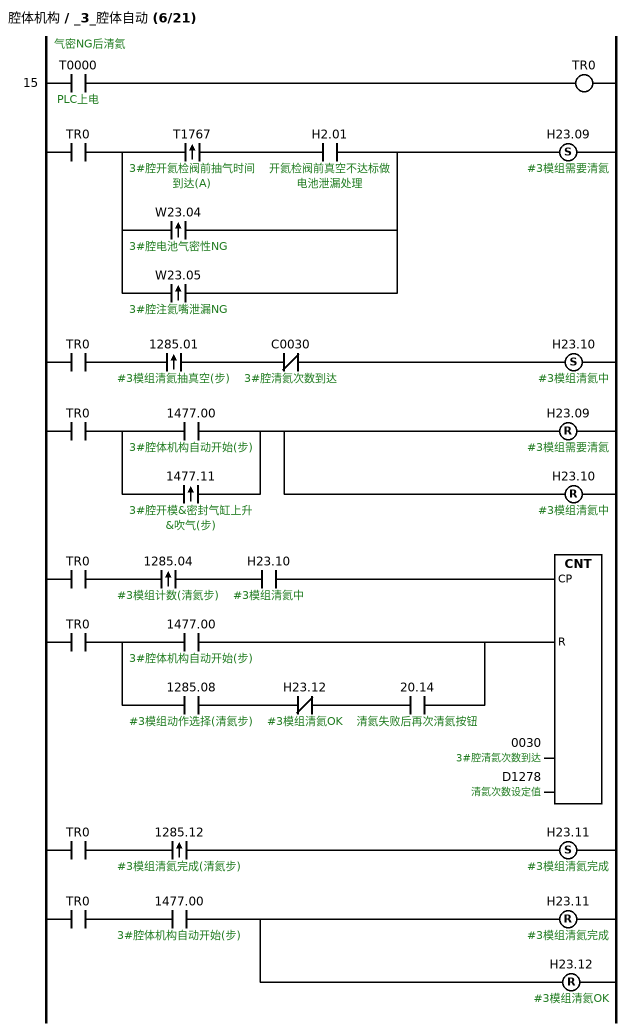
; rung 15: 气密NG后清氦
LD T0000  ; PLC上电
OUT TR0
@LD T1767  ; 3#腔开氦检阀前抽气时间到达(A)
AND H2.01  ; 开氦检阀前真空不达标做电池泄漏处理
@OR W23.04  ; 3#腔电池气密性NG
@OR W23.05  ; 3#腔注氦嘴泄漏NG
ANDLD
SET H23.09  ; #3模组需要清氦
LD TR0
@AND 1285.01  ; #3模组清氦抽真空(步)
ANDNOT C0030  ; 3#腔清氦次数到达
SET H23.10  ; #3模组清氦中
LD TR0
LD 1477.00  ; 3#腔体机构自动开始(步)
@OR 1477.11  ; 3#腔开模&密封气缸上升&吹气(步)
ANDLD
RSET H23.09  ; #3模组需要清氦
RSET H23.10  ; #3模组清氦中
LD TR0
@AND 1285.04  ; #3模组计数(清氦步)
AND H23.10  ; #3模组清氦中
LD TR0
LD 1477.00  ; 3#腔体机构自动开始(步)
LD 1285.08  ; #3模组动作选择(清氦步)
ANDNOT H23.12  ; #3模组清氦OK
AND 20.14  ; 清氦失败后再次清氦按钮
ORLD
ANDLD
CNT 0030 D1278  ; 清氦次数设定值, 3#腔清氦次数到达
LD TR0
@AND 1285.12  ; #3模组清氦完成(清氦步)
SET H23.11  ; #3模组清氦完成
LD TR0
AND 1477.00  ; 3#腔体机构自动开始(步)
RSET H23.11  ; #3模组清氦完成
RSET H23.12  ; #3模组清氦OK

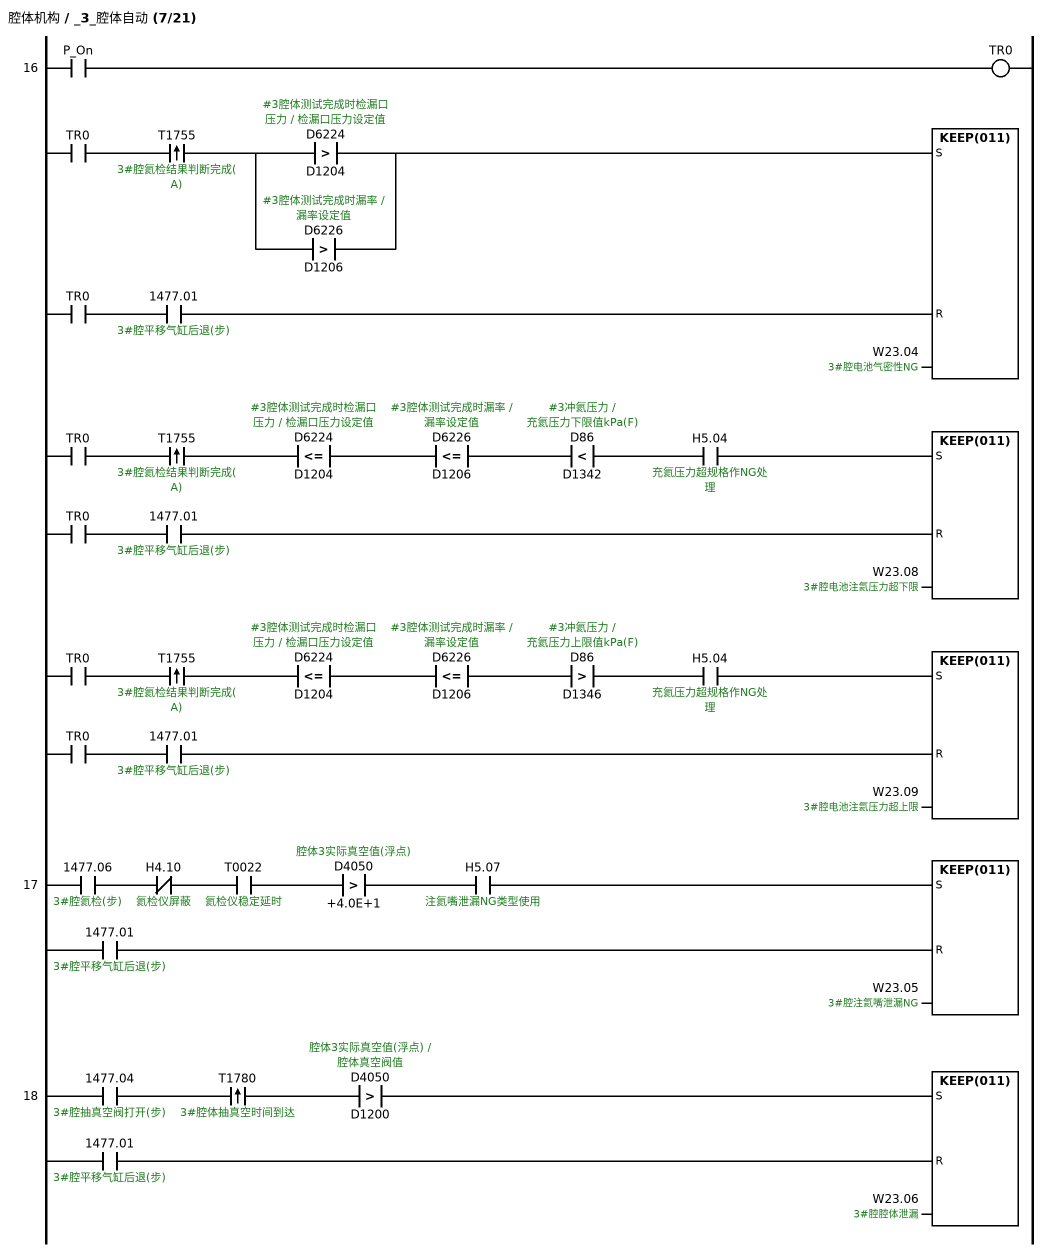
; rung 16
LD P_On
OUT TR0
@AND T1755  ; 3#腔氦检结果判断完成(A)
LD>F(333) D6224 D1204  ; #3腔体测试完成时检漏口压力, 检漏口压力设定值
OR>F(333) D6226 D1206  ; #3腔体测试完成时漏率, 漏率设定值
ANDLD
LD TR0
AND 1477.01  ; 3#腔平移气缸后退(步)
KEEP(011) W23.04  ; 3#腔电池气密性NG
LD TR0
@AND T1755  ; 3#腔氦检结果判断完成(A)
AND<=F(332) D6224 D1204  ; #3腔体测试完成时检漏口压力, 检漏口压力设定值
AND<=F(332) D6226 D1206  ; #3腔体测试完成时漏率, 漏率设定值
AND<F(331) D86 D1342  ; #3冲氦压力, 充氦压力下限值kPa(F)
AND H5.04  ; 充氦压力超规格作NG处理
LD TR0
AND 1477.01  ; 3#腔平移气缸后退(步)
KEEP(011) W23.08  ; 3#腔电池注氦压力超下限
LD TR0
@AND T1755  ; 3#腔氦检结果判断完成(A)
AND<=F(332) D6224 D1204  ; #3腔体测试完成时检漏口压力, 检漏口压力设定值
AND<=F(332) D6226 D1206  ; #3腔体测试完成时漏率, 漏率设定值
AND>F(333) D86 D1346  ; #3冲氦压力, 充氦压力上限值kPa(F)
AND H5.04  ; 充氦压力超规格作NG处理
LD TR0
AND 1477.01  ; 3#腔平移气缸后退(步)
KEEP(011) W23.09  ; 3#腔电池注氦压力超上限
; rung 17
LD 1477.06  ; 3#腔氦检(步)
ANDNOT H4.10  ; 氦检仪屏蔽
AND T0022  ; 氦检仪稳定延时
AND>F(333) D4050 +4.0E+1  ; 腔体3实际真空值(浮点)
AND H5.07  ; 注氦嘴泄漏NG类型使用
LD 1477.01  ; 3#腔平移气缸后退(步)
KEEP(011) W23.05  ; 3#腔注氦嘴泄漏NG
; rung 18
LD 1477.04  ; 3#腔抽真空阀打开(步)
@AND T1780  ; 3#腔体抽真空时间到达
AND>F(333) D4050 D1200  ; 腔体3实际真空值(浮点), 腔体真空阀值
LD 1477.01  ; 3#腔平移气缸后退(步)
KEEP(011) W23.06  ; 3#腔腔体泄漏

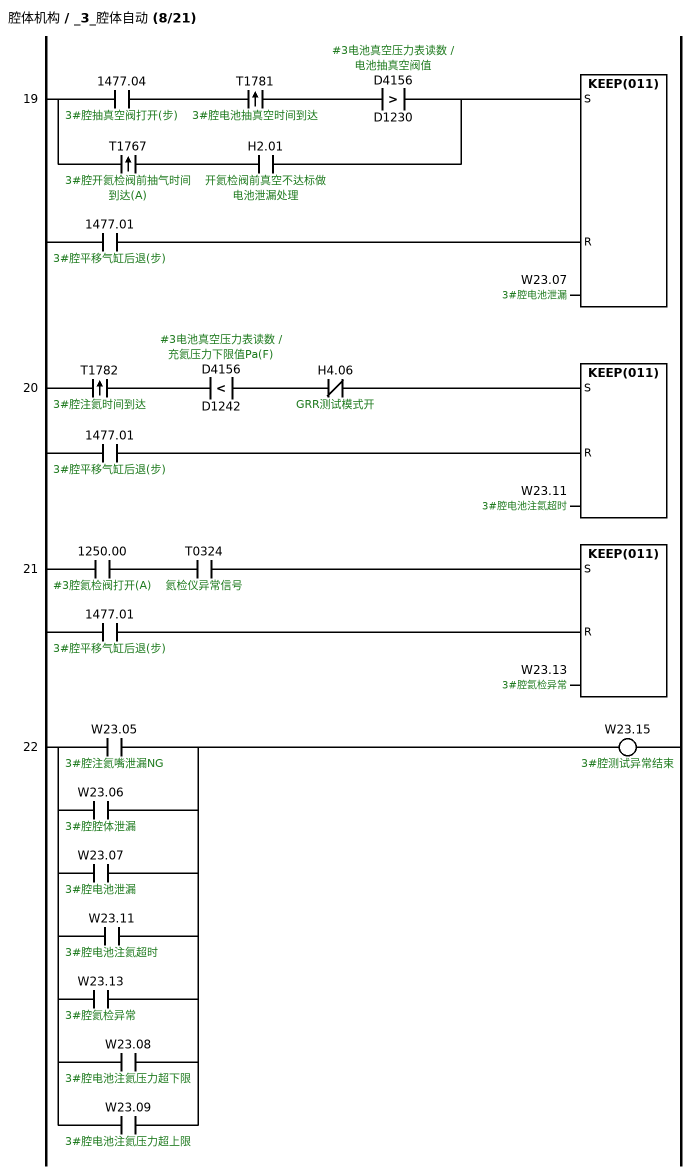
; rung 19
LD 1477.04  ; 3#腔抽真空阀打开(步)
@AND T1781  ; 3#腔电池抽真空时间到达
AND>F(333) D4156 D1230  ; #3电池真空压力表读数, 电池抽真空阀值
@LD T1767  ; 3#腔开氦检阀前抽气时间到达(A)
AND H2.01  ; 开氦检阀前真空不达标做电池泄漏处理
ORLD
LD 1477.01  ; 3#腔平移气缸后退(步)
KEEP(011) W23.07  ; 3#腔电池泄漏
; rung 20
@LD T1782  ; 3#腔注氦时间到达
AND<F(331) D4156 D1242  ; #3电池真空压力表读数, 充氦压力下限值Pa(F)
ANDNOT H4.06  ; GRR测试模式开
LD 1477.01  ; 3#腔平移气缸后退(步)
KEEP(011) W23.11  ; 3#腔电池注氦超时
; rung 21
LD 1250.00  ; #3腔氦检阀打开(A)
AND T0324  ; 氦检仪异常信号
LD 1477.01  ; 3#腔平移气缸后退(步)
KEEP(011) W23.13  ; 3#腔氦检异常
; rung 22
LD W23.05  ; 3#腔注氦嘴泄漏NG
OR W23.06  ; 3#腔腔体泄漏
OR W23.07  ; 3#腔电池泄漏
OR W23.11  ; 3#腔电池注氦超时
OR W23.13  ; 3#腔氦检异常
OR W23.08  ; 3#腔电池注氦压力超下限
OR W23.09  ; 3#腔电池注氦压力超上限
OUT W23.15  ; 3#腔测试异常结束

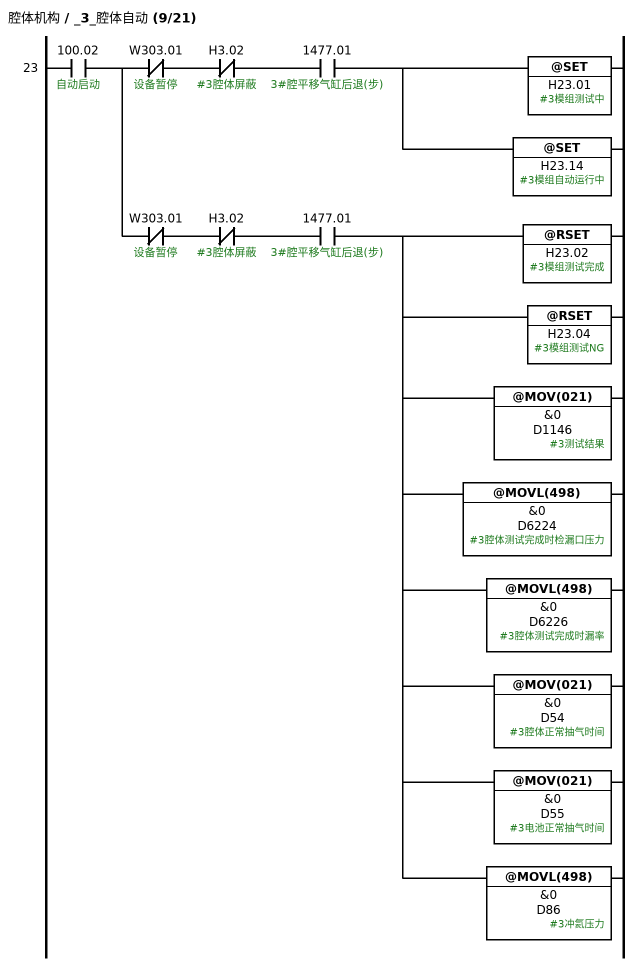
; rung 23
LD 100.02  ; 自动启动
OUT TR0
ANDNOT W303.01  ; 设备暂停
ANDNOT H3.02  ; #3腔体屏蔽
AND 1477.01  ; 3#腔平移气缸后退(步)
@SET H23.01  ; #3模组测试中
@SET H23.14  ; #3模组自动运行中
LD TR0
ANDNOT W303.01  ; 设备暂停
ANDNOT H3.02  ; #3腔体屏蔽
AND 1477.01  ; 3#腔平移气缸后退(步)
@RSET H23.02  ; #3模组测试完成
@RSET H23.04  ; #3模组测试NG
@MOV(021) &0 D1146  ; #3测试结果
@MOVL(498) &0 D6224  ; #3腔体测试完成时检漏口压力
@MOVL(498) &0 D6226  ; #3腔体测试完成时漏率
@MOV(021) &0 D54  ; #3腔体正常抽气时间
@MOV(021) &0 D55  ; #3电池正常抽气时间
@MOVL(498) &0 D86  ; #3冲氦压力

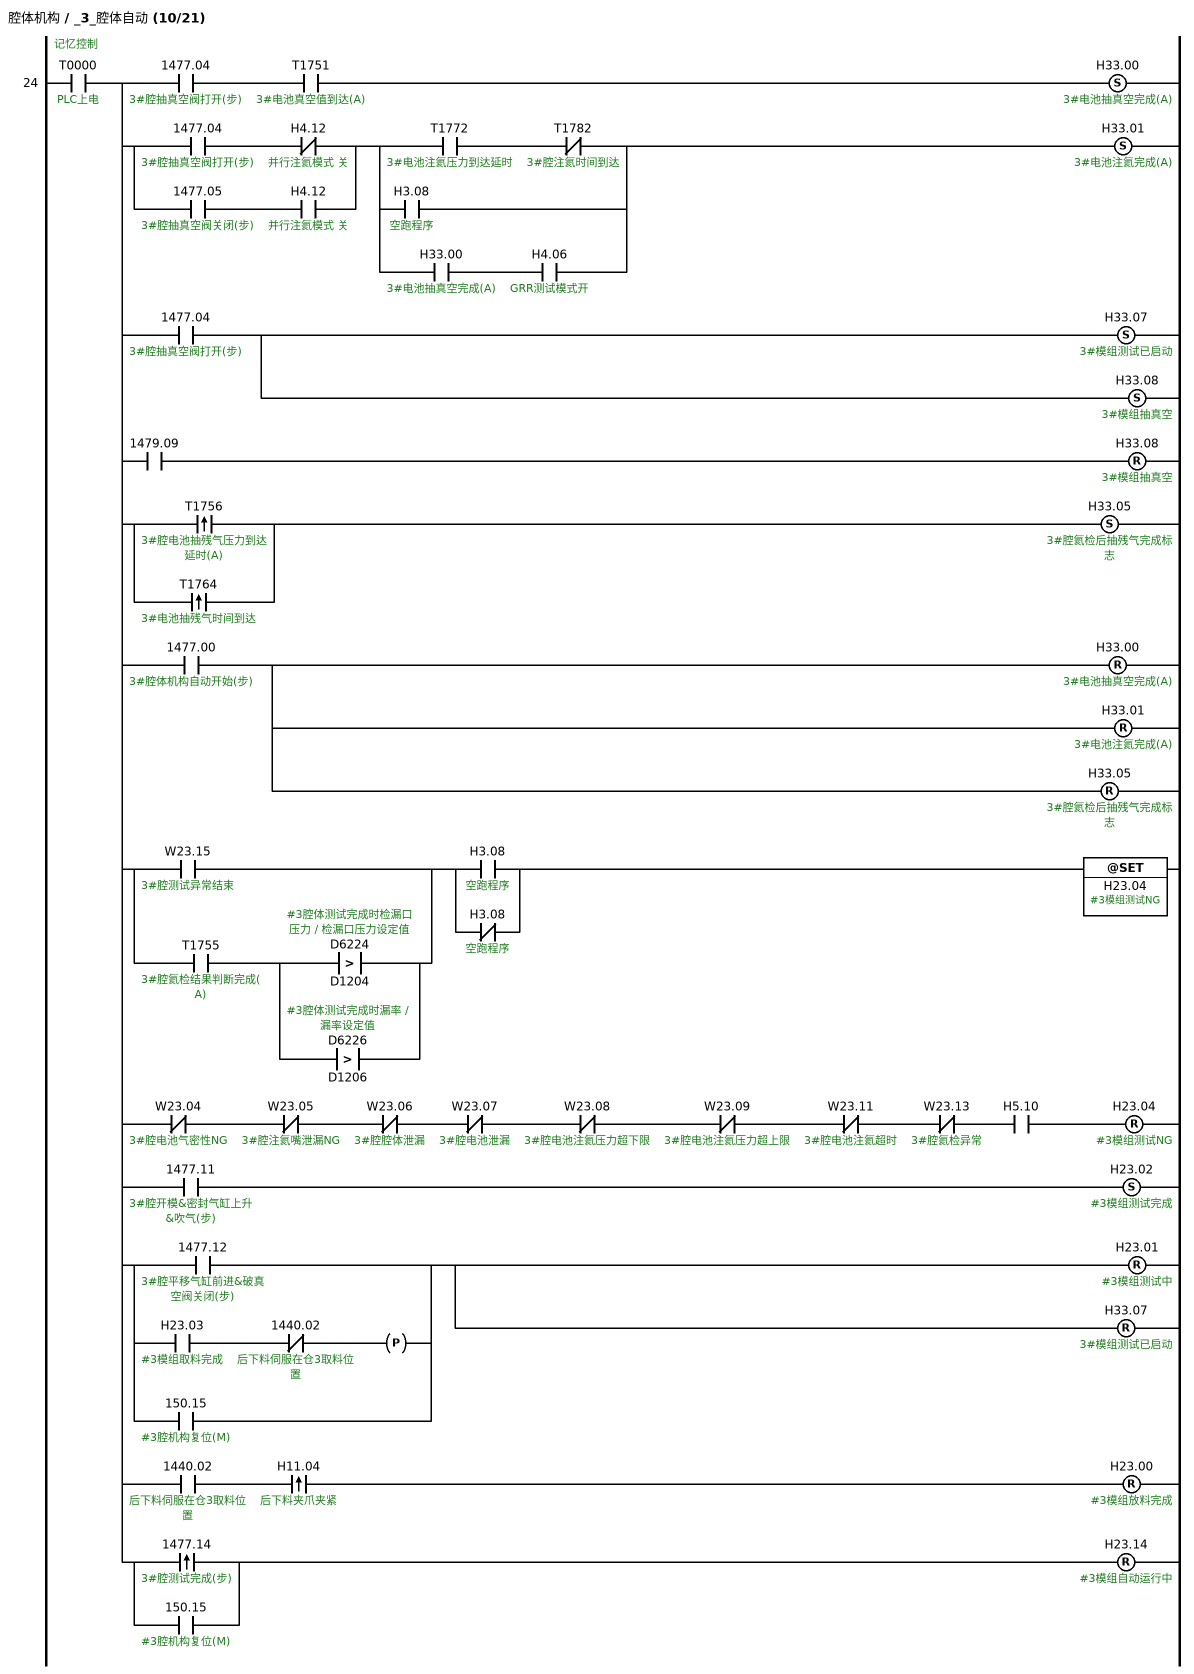
; rung 24: 记忆控制
LD T0000  ; PLC上电
OUT TR0
AND 1477.04  ; 3#腔抽真空阀打开(步)
AND T1751  ; 3#电池真空值到达(A)
SET H33.00  ; 3#电池抽真空完成(A)
LD TR0
LD 1477.04  ; 3#腔抽真空阀打开(步)
ANDNOT H4.12  ; 并行注氦模式 关
LD 1477.05  ; 3#腔抽真空阀关闭(步)
AND H4.12  ; 并行注氦模式 关
ORLD
ANDLD
LD T1772  ; 3#电池注氦压力到达延时
ANDNOT T1782  ; 3#腔注氦时间到达
OR H3.08  ; 空跑程序
LD H33.00  ; 3#电池抽真空完成(A)
AND H4.06  ; GRR测试模式开
ORLD
ANDLD
SET H33.01  ; 3#电池注氦完成(A)
LD TR0
AND 1477.04  ; 3#腔抽真空阀打开(步)
SET H33.07  ; 3#模组测试已启动
SET H33.08  ; 3#模组抽真空
LD TR0
AND 1479.09
RSET H33.08  ; 3#模组抽真空
LD TR0
@LD T1756  ; 3#腔电池抽残气压力到达延时(A)
@OR T1764  ; 3#电池抽残气时间到达
ANDLD
SET H33.05  ; 3#腔氦检后抽残气完成标志
LD TR0
AND 1477.00  ; 3#腔体机构自动开始(步)
RSET H33.00  ; 3#电池抽真空完成(A)
RSET H33.01  ; 3#电池注氦完成(A)
RSET H33.05  ; 3#腔氦检后抽残气完成标志
LD TR0
LD W23.15  ; 3#腔测试异常结束
LD T1755  ; 3#腔氦检结果判断完成(A)
LD>F(333) D6224 D1204  ; #3腔体测试完成时检漏口压力, 检漏口压力设定值
OR>F(333) D6226 D1206  ; #3腔体测试完成时漏率, 漏率设定值
ANDLD
ORLD
ANDLD
LD H3.08  ; 空跑程序
ORNOT H3.08  ; 空跑程序
ANDLD
@SET H23.04  ; #3模组测试NG
LD TR0
ANDNOT W23.04  ; 3#腔电池气密性NG
ANDNOT W23.05  ; 3#腔注氦嘴泄漏NG
ANDNOT W23.06  ; 3#腔腔体泄漏
ANDNOT W23.07  ; 3#腔电池泄漏
ANDNOT W23.08  ; 3#腔电池注氦压力超下限
ANDNOT W23.09  ; 3#腔电池注氦压力超上限
ANDNOT W23.11  ; 3#腔电池注氦超时
ANDNOT W23.13  ; 3#腔氦检异常
AND H5.10
RSET H23.04  ; #3模组测试NG
LD TR0
AND 1477.11  ; 3#腔开模&密封气缸上升&吹气(步)
SET H23.02  ; #3模组测试完成
LD TR0
LD 1477.12  ; 3#腔平移气缸前进&破真空阀关闭(步)
LD H23.03  ; #3模组取料完成
ANDNOT 1440.02  ; 后下料伺服在仓3取料位置
UP(521)
ORLD
OR 150.15  ; #3腔机构复位(M)
ANDLD
RSET H23.01  ; #3模组测试中
RSET H33.07  ; 3#模组测试已启动
LD TR0
AND 1440.02  ; 后下料伺服在仓3取料位置
@AND H11.04  ; 后下料夹爪夹紧
RSET H23.00  ; #3模组放料完成
LD TR0
@LD 1477.14  ; 3#腔测试完成(步)
OR 150.15  ; #3腔机构复位(M)
ANDLD
RSET H23.14  ; #3模组自动运行中

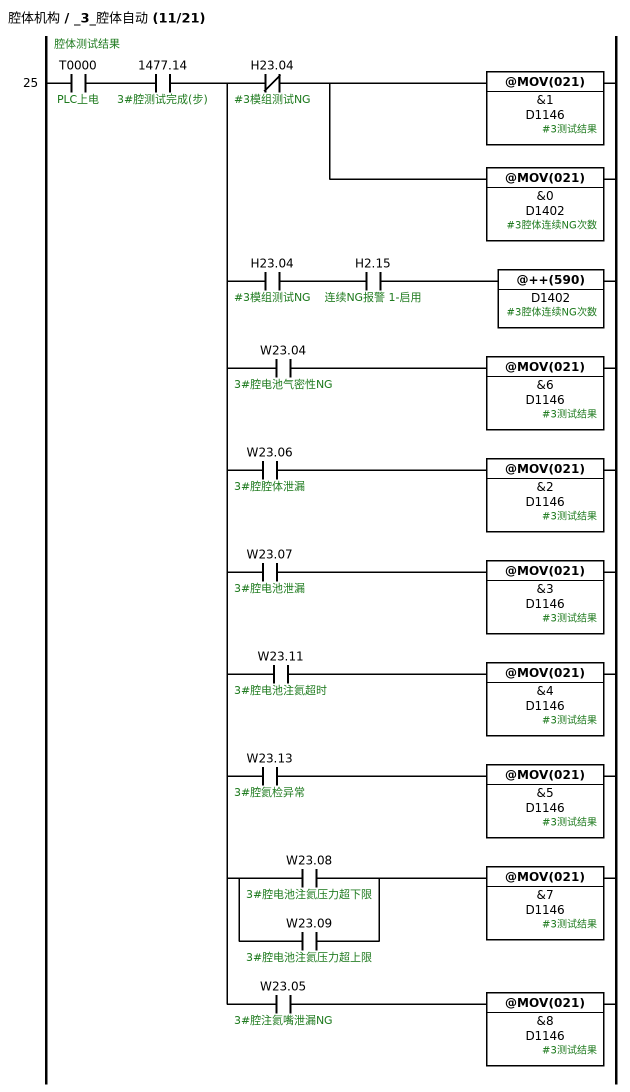
; rung 25: 腔体测试结果
LD T0000  ; PLC上电
AND 1477.14  ; 3#腔测试完成(步)
OUT TR0
ANDNOT H23.04  ; #3模组测试NG
@MOV(021) &1 D1146  ; #3测试结果
@MOV(021) &0 D1402  ; #3腔体连续NG次数
LD TR0
AND H23.04  ; #3模组测试NG
AND H2.15  ; 连续NG报警 1-启用
@++(590) D1402  ; #3腔体连续NG次数
LD TR0
AND W23.04  ; 3#腔电池气密性NG
@MOV(021) &6 D1146  ; #3测试结果
LD TR0
AND W23.06  ; 3#腔腔体泄漏
@MOV(021) &2 D1146  ; #3测试结果
LD TR0
AND W23.07  ; 3#腔电池泄漏
@MOV(021) &3 D1146  ; #3测试结果
LD TR0
AND W23.11  ; 3#腔电池注氦超时
@MOV(021) &4 D1146  ; #3测试结果
LD TR0
AND W23.13  ; 3#腔氦检异常
@MOV(021) &5 D1146  ; #3测试结果
LD TR0
LD W23.08  ; 3#腔电池注氦压力超下限
OR W23.09  ; 3#腔电池注氦压力超上限
ANDLD
@MOV(021) &7 D1146  ; #3测试结果
LD TR0
AND W23.05  ; 3#腔注氦嘴泄漏NG
@MOV(021) &8 D1146  ; #3测试结果

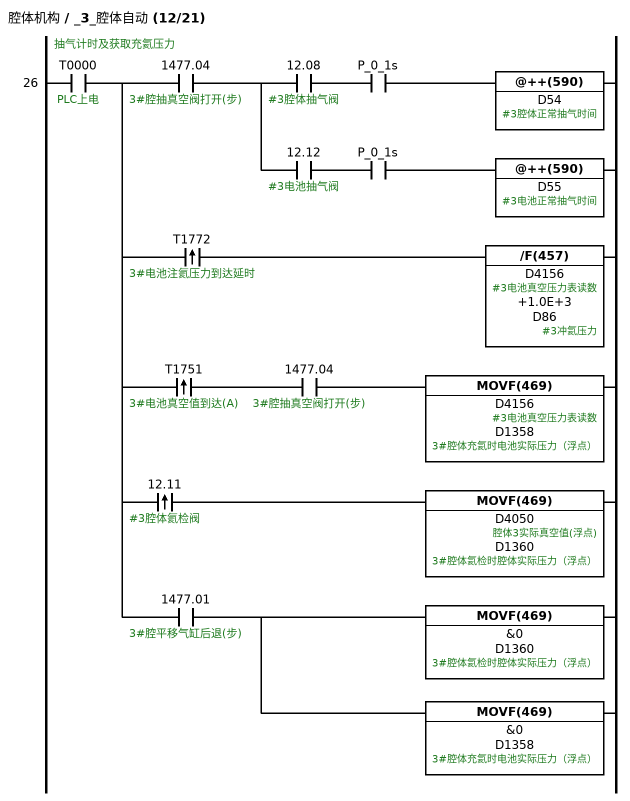
; rung 26: 抽气计时及获取充氦压力
LD T0000  ; PLC上电
OUT TR0
AND 1477.04  ; 3#腔抽真空阀打开(步)
OUT TR1
AND 12.08  ; #3腔体抽气阀
AND P_0_1s
@++(590) D54  ; #3腔体正常抽气时间
LD TR1
AND 12.12  ; #3电池抽气阀
AND P_0_1s
@++(590) D55  ; #3电池正常抽气时间
LD TR0
@AND T1772  ; 3#电池注氦压力到达延时
/F(457) D4156 +1.0E+3 D86  ; #3电池真空压力表读数, #3冲氦压力
LD TR0
@AND T1751  ; 3#电池真空值到达(A)
AND 1477.04  ; 3#腔抽真空阀打开(步)
MOVF(469) D4156 D1358  ; #3电池真空压力表读数, 3#腔体充氦时电池实际压力（浮点）
LD TR0
@AND 12.11  ; #3腔体氦检阀
MOVF(469) D4050 D1360  ; 腔体3实际真空值(浮点), 3#腔体氦检时腔体实际压力（浮点）
LD TR0
AND 1477.01  ; 3#腔平移气缸后退(步)
MOVF(469) &0 D1360  ; 3#腔体氦检时腔体实际压力（浮点）
MOVF(469) &0 D1358  ; 3#腔体充氦时电池实际压力（浮点）

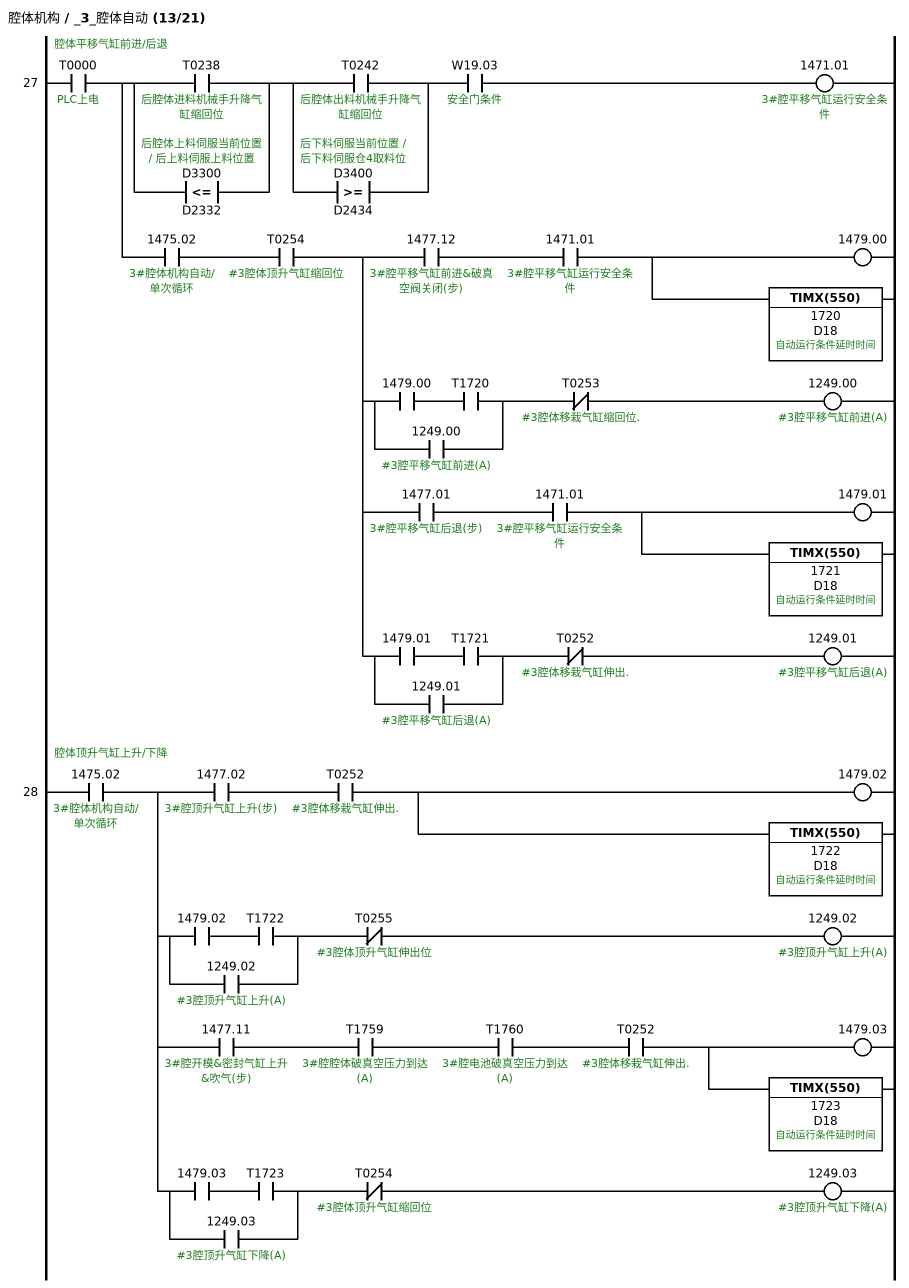
; rung 27: 腔体平移气缸前进/后退
LD T0000  ; PLC上电
OUT TR0
LD T0238  ; 后腔体进料机械手升降气缸缩回位
OR<=SL(318) D3300 D2332  ; 后腔体上料伺服当前位置, 后上料伺服上料位置
ANDLD
LD T0242  ; 后腔体出料机械手升降气缸缩回位
OR>=SL(328) D3400 D2434  ; 后下料伺服当前位置, 后下料伺服仓4取料位
ANDLD
AND W19.03  ; 安全门条件
OUT 1471.01  ; 3#腔平移气缸运行安全条件
LD TR0
AND 1475.02  ; 3#腔体机构自动/单次循环
AND T0254  ; #3腔体顶升气缸缩回位
OUT TR0
AND 1477.12  ; 3#腔平移气缸前进&破真空阀关闭(步)
AND 1471.01  ; 3#腔平移气缸运行安全条件
OUT 1479.00
TIMX(550) 1720 D18  ; 自动运行条件延时时间
LD TR0
LD 1479.00
AND T1720
OR 1249.00  ; #3腔平移气缸前进(A)
ANDLD
ANDNOT T0253  ; #3腔体移栽气缸缩回位.
OUT 1249.00  ; #3腔平移气缸前进(A)
LD TR0
AND 1477.01  ; 3#腔平移气缸后退(步)
AND 1471.01  ; 3#腔平移气缸运行安全条件
OUT 1479.01
TIMX(550) 1721 D18  ; 自动运行条件延时时间
LD TR0
LD 1479.01
AND T1721
OR 1249.01  ; #3腔平移气缸后退(A)
ANDLD
ANDNOT T0252  ; #3腔体移栽气缸伸出.
OUT 1249.01  ; #3腔平移气缸后退(A)
; rung 28: 腔体顶升气缸上升/下降
LD 1475.02  ; 3#腔体机构自动/单次循环
OUT TR0
AND 1477.02  ; 3#腔顶升气缸上升(步)
AND T0252  ; #3腔体移栽气缸伸出.
OUT 1479.02
TIMX(550) 1722 D18  ; 自动运行条件延时时间
LD TR0
LD 1479.02
AND T1722
OR 1249.02  ; #3腔顶升气缸上升(A)
ANDLD
ANDNOT T0255  ; #3腔体顶升气缸伸出位
OUT 1249.02  ; #3腔顶升气缸上升(A)
LD TR0
AND 1477.11  ; 3#腔开模&密封气缸上升&吹气(步)
AND T1759  ; 3#腔腔体破真空压力到达(A)
AND T1760  ; 3#腔电池破真空压力到达(A)
AND T0252  ; #3腔体移栽气缸伸出.
OUT 1479.03
TIMX(550) 1723 D18  ; 自动运行条件延时时间
LD TR0
LD 1479.03
AND T1723
OR 1249.03  ; #3腔顶升气缸下降(A)
ANDLD
ANDNOT T0254  ; #3腔体顶升气缸缩回位
OUT 1249.03  ; #3腔顶升气缸下降(A)

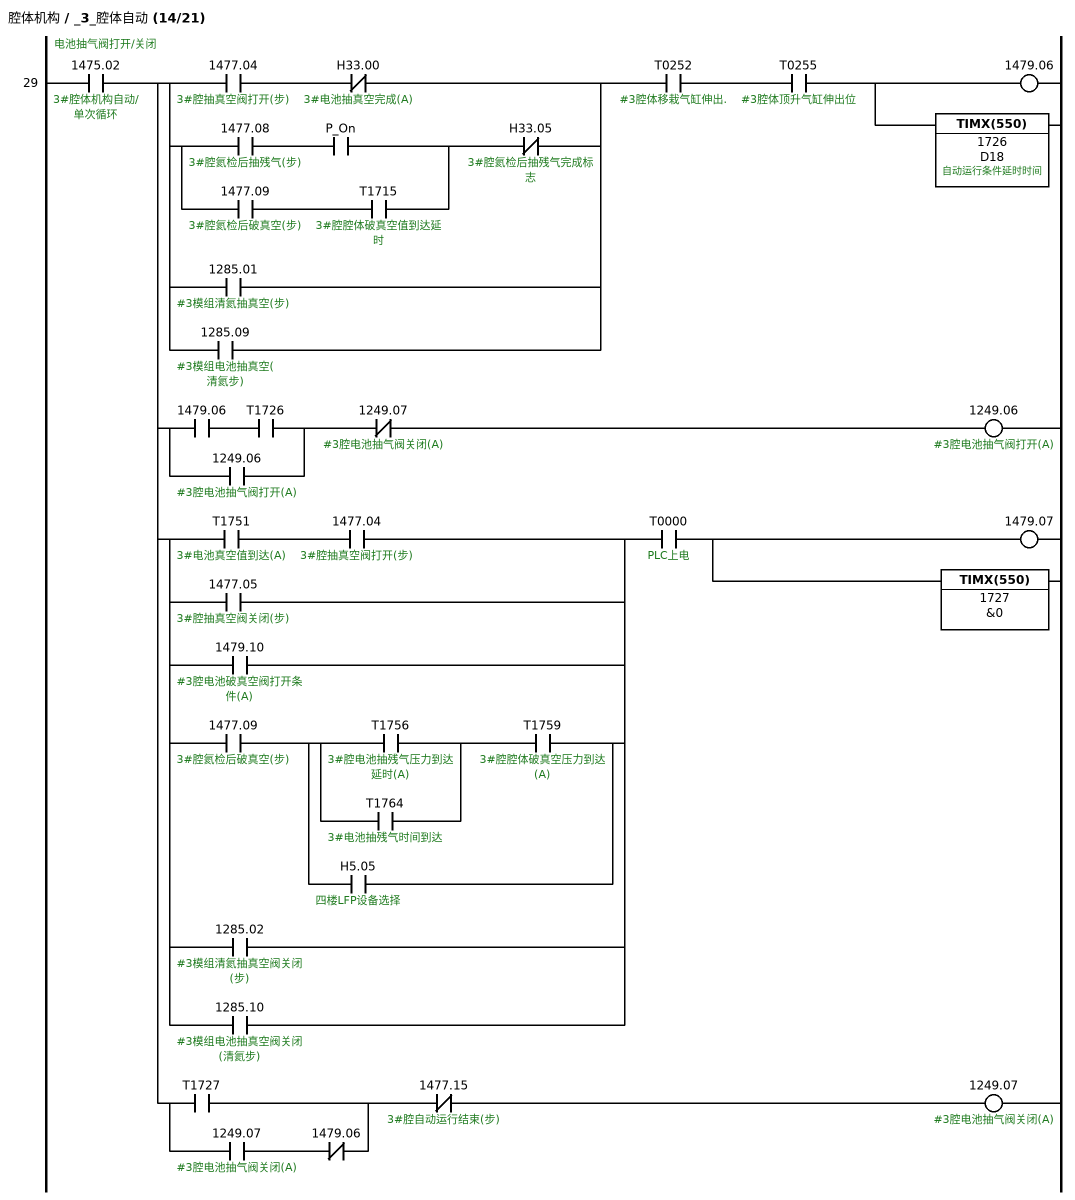
; rung 29: 电池抽气阀打开/关闭
LD 1475.02  ; 3#腔体机构自动/单次循环
OUT TR0
LD 1477.04  ; 3#腔抽真空阀打开(步)
ANDNOT H33.00  ; 3#电池抽真空完成(A)
LD 1477.08  ; 3#腔氦检后抽残气(步)
AND P_On
LD 1477.09  ; 3#腔氦检后破真空(步)
AND T1715  ; 3#腔腔体破真空值到达延时
ORLD
ANDNOT H33.05  ; 3#腔氦检后抽残气完成标志
ORLD
OR 1285.01  ; #3模组清氦抽真空(步)
OR 1285.09  ; #3模组电池抽真空(清氦步)
ANDLD
AND T0252  ; #3腔体移栽气缸伸出.
AND T0255  ; #3腔体顶升气缸伸出位
OUT 1479.06
TIMX(550) 1726 D18  ; 自动运行条件延时时间
LD TR0
LD 1479.06
AND T1726
OR 1249.06  ; #3腔电池抽气阀打开(A)
ANDLD
ANDNOT 1249.07  ; #3腔电池抽气阀关闭(A)
OUT 1249.06  ; #3腔电池抽气阀打开(A)
LD TR0
LD T1751  ; 3#电池真空值到达(A)
AND 1477.04  ; 3#腔抽真空阀打开(步)
OR 1477.05  ; 3#腔抽真空阀关闭(步)
OR 1479.10  ; #3腔电池破真空阀打开条件(A)
LD 1477.09  ; 3#腔氦检后破真空(步)
LD T1756  ; 3#腔电池抽残气压力到达延时(A)
OR T1764  ; 3#电池抽残气时间到达
AND T1759  ; 3#腔腔体破真空压力到达(A)
OR H5.05  ; 四楼LFP设备选择
ANDLD
ORLD
OR 1285.02  ; #3模组清氦抽真空阀关闭(步)
OR 1285.10  ; #3模组电池抽真空阀关闭(清氦步)
ANDLD
AND T0000  ; PLC上电
OUT 1479.07
TIMX(550) 1727 &0
LD TR0
LD T1727
LD 1249.07  ; #3腔电池抽气阀关闭(A)
ANDNOT 1479.06
ORLD
ANDLD
ANDNOT 1477.15  ; 3#腔自动运行结束(步)
OUT 1249.07  ; #3腔电池抽气阀关闭(A)

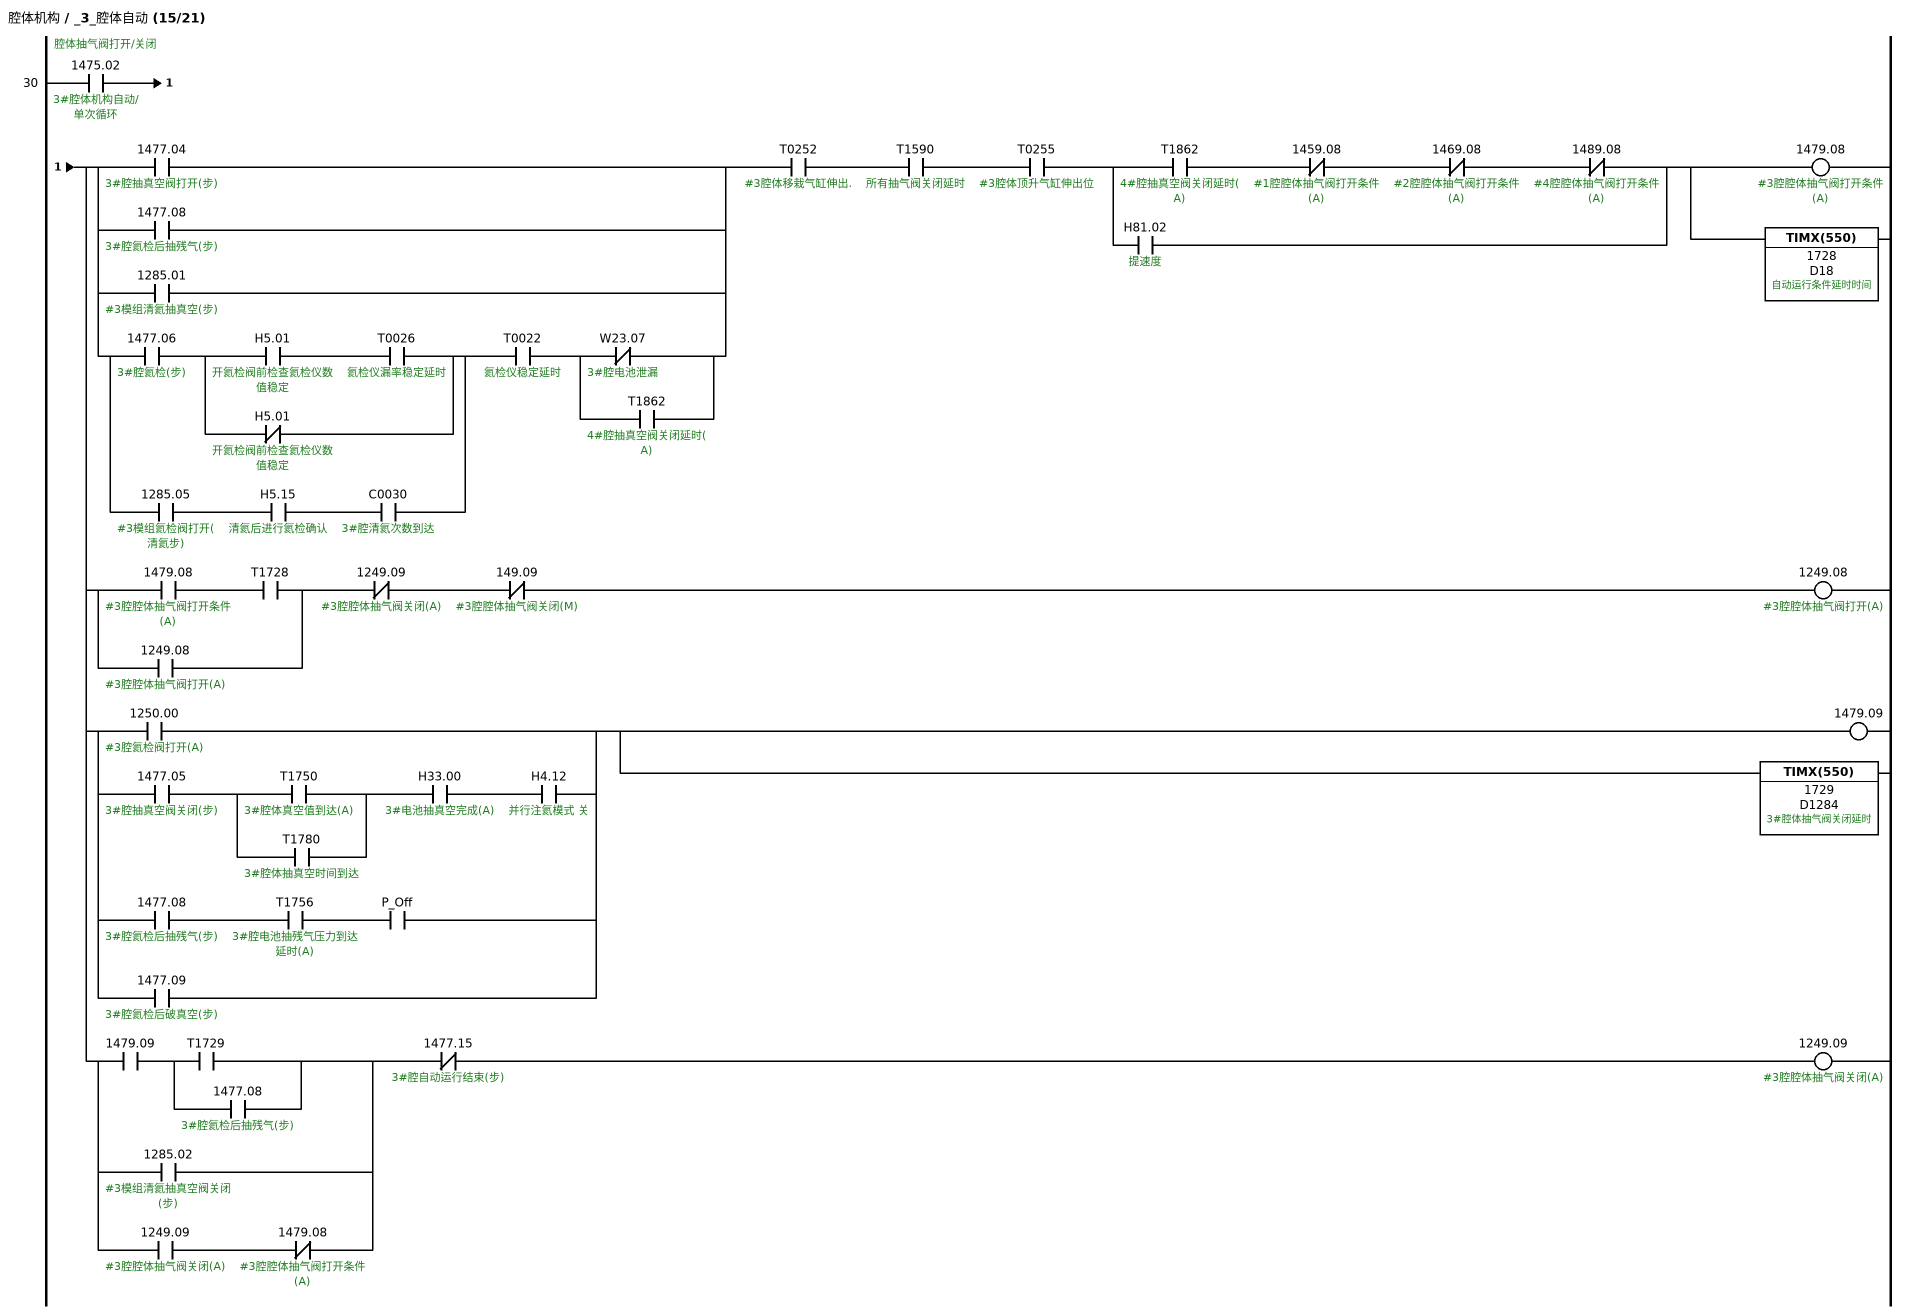
; rung 30: 腔体抽气阀打开/关闭
LD 1475.02  ; 3#腔体机构自动/单次循环
OUT TR0
LD 1477.04  ; 3#腔抽真空阀打开(步)
OR 1477.08  ; 3#腔氦检后抽残气(步)
OR 1285.01  ; #3模组清氦抽真空(步)
LD 1477.06  ; 3#腔氦检(步)
LD H5.01  ; 开氦检阀前检查氦检仪数值稳定
AND T0026  ; 氦检仪漏率稳定延时
ORNOT H5.01  ; 开氦检阀前检查氦检仪数值稳定
ANDLD
LD 1285.05  ; #3模组氦检阀打开(清氦步)
AND H5.15  ; 清氦后进行氦检确认
AND C0030  ; 3#腔清氦次数到达
ORLD
AND T0022  ; 氦检仪稳定延时
LDNOT W23.07  ; 3#腔电池泄漏
OR T1862  ; 4#腔抽真空阀关闭延时(A)
ANDLD
ORLD
ANDLD
AND T0252  ; #3腔体移栽气缸伸出.
AND T1590  ; 所有抽气阀关闭延时
AND T0255  ; #3腔体顶升气缸伸出位
LD T1862  ; 4#腔抽真空阀关闭延时(A)
ANDNOT 1459.08  ; #1腔腔体抽气阀打开条件(A)
ANDNOT 1469.08  ; #2腔腔体抽气阀打开条件(A)
ANDNOT 1489.08  ; #4腔腔体抽气阀打开条件(A)
OR H81.02  ; 提速度
ANDLD
OUT 1479.08  ; #3腔腔体抽气阀打开条件(A)
TIMX(550) 1728 D18  ; 自动运行条件延时时间
LD TR0
LD 1479.08  ; #3腔腔体抽气阀打开条件(A)
AND T1728
OR 1249.08  ; #3腔腔体抽气阀打开(A)
ANDLD
ANDNOT 1249.09  ; #3腔腔体抽气阀关闭(A)
ANDNOT 149.09  ; #3腔腔体抽气阀关闭(M)
OUT 1249.08  ; #3腔腔体抽气阀打开(A)
LD TR0
LD 1250.00  ; #3腔氦检阀打开(A)
LD 1477.05  ; 3#腔抽真空阀关闭(步)
LD T1750  ; 3#腔体真空值到达(A)
OR T1780  ; 3#腔体抽真空时间到达
ANDLD
AND H33.00  ; 3#电池抽真空完成(A)
AND H4.12  ; 并行注氦模式 关
ORLD
LD 1477.08  ; 3#腔氦检后抽残气(步)
AND T1756  ; 3#腔电池抽残气压力到达延时(A)
AND P_Off
ORLD
OR 1477.09  ; 3#腔氦检后破真空(步)
ANDLD
OUT 1479.09
TIMX(550) 1729 D1284  ; 3#腔体抽气阀关闭延时
LD TR0
LD 1479.09
LD T1729
OR 1477.08  ; 3#腔氦检后抽残气(步)
ANDLD
OR 1285.02  ; #3模组清氦抽真空阀关闭(步)
LD 1249.09  ; #3腔腔体抽气阀关闭(A)
ANDNOT 1479.08  ; #3腔腔体抽气阀打开条件(A)
ORLD
ANDLD
ANDNOT 1477.15  ; 3#腔自动运行结束(步)
OUT 1249.09  ; #3腔腔体抽气阀关闭(A)

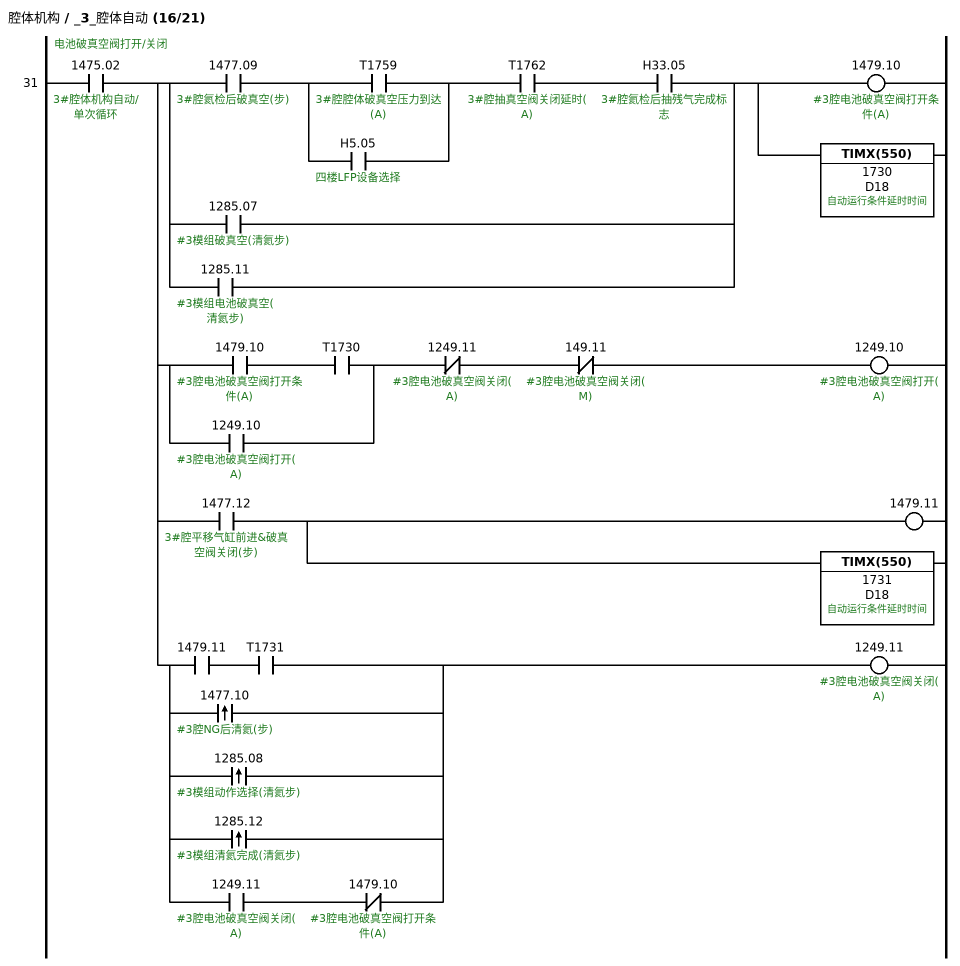
; rung 31: 电池破真空阀打开/关闭
LD 1475.02  ; 3#腔体机构自动/单次循环
OUT TR0
LD 1477.09  ; 3#腔氦检后破真空(步)
LD T1759  ; 3#腔腔体破真空压力到达(A)
OR H5.05  ; 四楼LFP设备选择
ANDLD
AND T1762  ; 3#腔抽真空阀关闭延时(A)
AND H33.05  ; 3#腔氦检后抽残气完成标志
OR 1285.07  ; #3模组破真空(清氦步)
OR 1285.11  ; #3模组电池破真空(清氦步)
ANDLD
OUT 1479.10  ; #3腔电池破真空阀打开条件(A)
TIMX(550) 1730 D18  ; 自动运行条件延时时间
LD TR0
LD 1479.10  ; #3腔电池破真空阀打开条件(A)
AND T1730
OR 1249.10  ; #3腔电池破真空阀打开(A)
ANDLD
ANDNOT 1249.11  ; #3腔电池破真空阀关闭(A)
ANDNOT 149.11  ; #3腔电池破真空阀关闭(M)
OUT 1249.10  ; #3腔电池破真空阀打开(A)
LD TR0
AND 1477.12  ; 3#腔平移气缸前进&破真空阀关闭(步)
OUT 1479.11
TIMX(550) 1731 D18  ; 自动运行条件延时时间
LD TR0
LD 1479.11
AND T1731
@OR 1477.10  ; #3腔NG后清氦(步)
@OR 1285.08  ; #3模组动作选择(清氦步)
@OR 1285.12  ; #3模组清氦完成(清氦步)
LD 1249.11  ; #3腔电池破真空阀关闭(A)
ANDNOT 1479.10  ; #3腔电池破真空阀打开条件(A)
ORLD
ANDLD
OUT 1249.11  ; #3腔电池破真空阀关闭(A)

